LIN {X 0,Y 361.99,Z 158.394,A -85,B 0,C 180,E1 -12970.064,E2 -12970.064} C_VEL
LIN {X 0,Y 361.976,Z 158.397,A -85,B 0,C 180,E1 -12973.887,E2 -12973.887} C_VEL
LIN {X 0,Y 361.88,Z 158.406,A -85,B 0,C 180,E1 -12978.104,E2 -12978.104} C_VEL
LIN {X 0,Y 361.849,Z 158.413,A -85,B 0,C 180,E1 -12981.656,E2 -12981.656} C_VEL
LIN {X 0,Y 361.849,Z 158.412,A -85,B 0,C 180,E1 -12985.296,E2 -12985.296} C_VEL
LIN {X 0,Y 361.853,Z 158.41,A -85,B 0,C 180,E1 -12989.074,E2 -12989.074} C_VEL
LIN {X 0,Y 361.845,Z 158.411,A -85,B 0,C 180,E1 -12992.946,E2 -12992.946} C_VEL
LIN {X 0,Y 361.861,Z 158.409,A -85,B 0,C 180,E1 -12995.638,E2 -12995.638} C_VEL
LIN {X 0,Y 361.823,Z 158.416,A -85,B 0,C 180,E1 -12999.018,E2 -12999.018} C_VEL
LIN {X 0,Y 361.828,Z 158.414,A -85,B 0,C 180,E1 -13002.831,E2 -13002.831} C_VEL
LIN {X 0,Y 361.812,Z 158.413,A -85,B 0,C 180,E1 -13005.948,E2 -13005.948} C_VEL
LIN {X 0,Y 361.81,Z 158.416,A -85,B 0,C 180,E1 -13009.25,E2 -13009.25} C_VEL
LIN {X 0,Y 361.861,Z 158.412,A -85,B 0,C 180,E1 -13012.982,E2 -13012.982} C_VEL
LIN {X 0,Y 361.858,Z 158.412,A -85,B 0,C 180,E1 -13016.632,E2 -13016.632} C_VEL
LIN {X 0,Y 361.865,Z 158.409,A -85,B 0,C 180,E1 -13020.315,E2 -13020.315} C_VEL
LIN {X 0,Y 361.868,Z 158.547,A -85,B 0,C 180,E1 -13020.81,E2 -13020.81} C_VEL
LIN {X 0,Y 364.371,Z 170.848,A -85,B 0,C 180,E1 -13023.973,E2 -13023.973} C_VEL
LIN {X 0,Y 365.33,Z 177.294,A -85,B 0,C 180,E1 -13025.569,E2 -13025.569} C_VEL
LIN {X 0,Y 364.23,Z 189.968,A -85,B 0,C 180,E1 -13028.493,E2 -13028.493} C_VEL
LIN {X 0,Y 369.048,Z 223.646,A -85,B 0,C 180,E1 -13029.496,E2 -13029.496} C_VEL
LIN {X 0,Y 367.536,Z 298.731,A -85,B 0,C 180,E1 -13031.102,E2 -13031.102} C_VEL
LIN {X 0,Y 366.947,Z 312.235,A -85,B 0,C 180,E1 -13031.614,E2 -13031.614} C_VEL
LIN {X 0,Y 366.191,Z 324.024,A -85,B 0,C 180,E1 -13032.261,E2 -13032.261} C_VEL
LIN {X 0,Y 365.354,Z 335.279,A -85,B 0,C 180,E1 -13033.085,E2 -13033.085} C_VEL
LIN {X 0,Y 364.275,Z 346.955,A -85,B 0,C 180,E1 -13034.186,E2 -13034.186} C_VEL
LIN {X 0,Y 363.436,Z 357.505,A -85,B 0,C 180,E1 -13035.44,E2 -13035.44} C_VEL
LIN {X 0,Y 362.593,Z 366.984,A -85,B 0,C 180,E1 -13036.836,E2 -13036.836} C_VEL
LIN {X 0,Y 361.669,Z 376.126,A -85,B 0,C 180,E1 -13038.511,E2 -13038.511} C_VEL
LIN {X 0,Y 361.112,Z 383.491,A -85,B 0,C 180,E1 -13040.195,E2 -13040.195} C_VEL
LIN {X 0,Y 360.759,Z 388.451,A -85,B 0,C 180,E1 -13041.598,E2 -13041.598} C_VEL
LIN {X 0,Y 360.499,Z 393.254,A -85,B 0,C 180,E1 -13043.283,E2 -13043.283} C_VEL
LIN {X 0,Y 360.345,Z 396.905,A -85,B 0,C 180,E1 -13044.965,E2 -13044.965} C_VEL
LIN {X 0,Y 360.301,Z 399.51,A -85,B 0,C 180,E1 -13046.645,E2 -13046.645} C_VEL
LIN {X 0,Y 360.266,Z 400.723,A -85,B 0,C 180,E1 -13047.764,E2 -13047.764} C_VEL
LIN {X 0,Y 360.319,Z 401.482,A -85,B 0,C 180,E1 -13048.882,E2 -13048.882} C_VEL
LIN {X 0,Y 360.361,Z 401.829,A -85,B 0,C 180,E1 -13050,E2 -13050} C_VEL
LIN {X 0,Y 360.303,Z 401.777,A -85,B 0,C 180,E1 -13051.117,E2 -13051.117} C_VEL
LIN {X 0,Y 360.263,Z 401.326,A -85,B 0,C 180,E1 -13052.236,E2 -13052.236} C_VEL
LIN {X 0,Y 360.297,Z 400.429,A -85,B 0,C 180,E1 -13053.355,E2 -13053.355} C_VEL
LIN {X 0,Y 360.346,Z 399.119,A -85,B 0,C 180,E1 -13054.474,E2 -13054.474} C_VEL
LIN {X 0,Y 360.379,Z 396.74,A -85,B 0,C 180,E1 -13055.961,E2 -13055.961} C_VEL
LIN {X 0,Y 360.69,Z 392.557,A -85,B 0,C 180,E1 -13057.839,E2 -13057.839} C_VEL
LIN {X 0,Y 361.118,Z 387.637,A -85,B 0,C 180,E1 -13059.522,E2 -13059.522} C_VEL
LIN {X 0,Y 361.758,Z 381.447,A -85,B 0,C 180,E1 -13061.202,E2 -13061.202} C_VEL
LIN {X 0,Y 362.725,Z 373.766,A -85,B 0,C 180,E1 -13062.874,E2 -13062.874} C_VEL
LIN {X 0,Y 363.683,Z 365.931,A -85,B 0,C 180,E1 -13064.263,E2 -13064.263} C_VEL
LIN {X 0,Y 364.646,Z 356.392,A -85,B 0,C 180,E1 -13065.654,E2 -13065.654} C_VEL
LIN {X 0,Y 365.843,Z 345.844,A -85,B 0,C 180,E1 -13066.891,E2 -13066.891} C_VEL
LIN {X 0,Y 367.109,Z 334.15,A -85,B 0,C 180,E1 -13067.98,E2 -13067.98} C_VEL
LIN {X 0,Y 368.232,Z 321.75,A -85,B 0,C 180,E1 -13068.86,E2 -13068.86} C_VEL
LIN {X 0,Y 369.141,Z 308.873,A -85,B 0,C 180,E1 -13069.534,E2 -13069.534} C_VEL
LIN {X 0,Y 369.816,Z 296.528,A -85,B 0,C 180,E1 -13069.967,E2 -13069.967} C_VEL
LIN {X 0,Y 371.47,Z 222.319,A -85,B 0,C 180,E1 -13071.596,E2 -13071.596} C_VEL
LIN {X 0,Y 368.034,Z 201.179,A -85,B 0,C 180,E1 -13072.355,E2 -13072.355} C_VEL
LIN {X 0,Y 365.368,Z 188.435,A -85,B 0,C 180,E1 -13072.904,E2 -13072.904} C_VEL
LIN {X 0,Y 366.207,Z 179.523,A -85,B 0,C 180,E1 -13074.974,E2 -13074.974} C_VEL
LIN {X 0,Y 364.952,Z 172.094,A -85,B 0,C 180,E1 -13076.897,E2 -13076.897} C_VEL
LIN {X 0,Y 362.672,Z 161.769,A -85,B 0,C 180,E1 -13079.712,E2 -13079.712} C_VEL
LIN {X 0,Y 361.872,Z 158.417,A -85,B 0,C 180,E1 -13080.707,E2 -13080.707} C_VEL
LIN {X 0,Y 361.849,Z 158.412,A -85,B 0,C 180,E1 -13084.28,E2 -13084.28} C_VEL
LIN {X 0,Y 361.855,Z 158.414,A -85,B 0,C 180,E1 -13087.22,E2 -13087.22} C_VEL
LIN {X 0,Y 361.808,Z 158.419,A -85,B 0,C 180,E1 -13090.75,E2 -13090.75} C_VEL
LIN {X 0,Y 361.809,Z 158.42,A -85,B 0,C 180,E1 -13094.369,E2 -13094.369} C_VEL
LIN {X 0,Y 361.819,Z 158.411,A -85,B 0,C 180,E1 -13097.57,E2 -13097.57} C_VEL
LIN {X 0,Y 361.838,Z 158.412,A -85,B 0,C 180,E1 -13101.571,E2 -13101.571} C_VEL
LIN {X 0,Y 361.866,Z 158.409,A -85,B 0,C 180,E1 -13104.656,E2 -13104.656} C_VEL
LIN {X 0,Y 361.833,Z 158.413,A -85,B 0,C 180,E1 -13108.37,E2 -13108.37} C_VEL
LIN {X 0,Y 361.845,Z 158.41,A -85,B 0,C 180,E1 -13110.95,E2 -13110.95} C_VEL
LIN {X 0,Y 361.855,Z 158.409,A -85,B 0,C 180,E1 -13114.704,E2 -13114.704} C_VEL
LIN {X 0,Y 361.847,Z 158.408,A -85,B 0,C 180,E1 -13118.344,E2 -13118.344} C_VEL
LIN {X 0,Y 361.89,Z 158.402,A -85,B 0,C 180,E1 -13122.097,E2 -13122.097} C_VEL
LIN {X 0,Y 361.974,Z 158.395,A -85,B 0,C 180,E1 -13126.113,E2 -13126.113} C_VEL
LIN {X 0,Y 361.988,Z 158.395,A -85,B 0,C 180,E1 -13129.936,E2 -13129.936} C_VEL
LIN {X 0,Y 362.111,Z 158.378,A -85,B 0,C 180,E1 -13133.312,E2 -13133.312} C_VEL
LIN {X 0,Y 362.256,Z 158.359,A -85,B 0,C 180,E1 -13137.776,E2 -13137.776} C_VEL
LIN {X 0,Y 362.166,Z 158.367,A -85,B 0,C 180,E1 -13141.111,E2 -13141.111} C_VEL
LIN {X 0,Y 362.256,Z 158.362,A -85,B 0,C 180,E1 -13142.223,E2 -13142.223} C_VEL
LIN {X 0,Y 362.111,Z 158.379,A -85,B 0,C 180,E1 -13146.687,E2 -13146.687} C_VEL
LIN {X 0,Y 361.987,Z 158.399,A -85,B 0,C 180,E1 -13150.063,E2 -13150.063} C_VEL
LIN {X 0,Y 361.972,Z 158.404,A -85,B 0,C 180,E1 -13153.886,E2 -13153.886} C_VEL
LIN {X 0,Y 361.928,Z 158.506,A -85,B 0,C 180,E1 -13157.348,E2 -13157.348} C_VEL
LIN {X 0,Y 364.483,Z 169.841,A -85,B 0,C 180,E1 -13160.603,E2 -13160.603} C_VEL
LIN {X 0,Y 364.864,Z 171.752,A -85,B 0,C 180,E1 -13161.134,E2 -13161.134} C_VEL
LIN {X 0,Y 368.482,Z 181.215,A -85,B 0,C 180,E1 -13161.661,E2 -13161.661} C_VEL
LIN {X 0,Y 372.141,Z 198.437,A -85,B 0,C 180,E1 -13162.349,E2 -13162.349} C_VEL
LIN {X 0,Y 370.023,Z 279.828,A -85,B 0,C 180,E1 -13164.135,E2 -13164.135} C_VEL
LIN {X 0,Y 369.348,Z 293.268,A -85,B 0,C 180,E1 -13164.651,E2 -13164.651} C_VEL
LIN {X 0,Y 368.609,Z 305.305,A -85,B 0,C 180,E1 -13165.327,E2 -13165.327} C_VEL
LIN {X 0,Y 367.629,Z 317.028,A -85,B 0,C 180,E1 -13166.207,E2 -13166.207} C_VEL
LIN {X 0,Y 366.407,Z 329.368,A -85,B 0,C 180,E1 -13167.409,E2 -13167.409} C_VEL
LIN {X 0,Y 365.378,Z 338.355,A -85,B 0,C 180,E1 -13168.501,E2 -13168.501} C_VEL
LIN {X 0,Y 364.251,Z 347.761,A -85,B 0,C 180,E1 -13169.901,E2 -13169.901} C_VEL
LIN {X 0,Y 363.096,Z 356.944,A -85,B 0,C 180,E1 -13171.61,E2 -13171.61} C_VEL
LIN {X 0,Y 362.288,Z 363.667,A -85,B 0,C 180,E1 -13173.166,E2 -13173.166} C_VEL
LIN {X 0,Y 361.625,Z 369.267,A -85,B 0,C 180,E1 -13174.77,E2 -13174.77} C_VEL
LIN {X 0,Y 361.125,Z 373.689,A -85,B 0,C 180,E1 -13176.363,E2 -13176.363} C_VEL
LIN {X 0,Y 360.619,Z 378.205,A -85,B 0,C 180,E1 -13178.582,E2 -13178.582} C_VEL
LIN {X 0,Y 360.314,Z 380.682,A -85,B 0,C 180,E1 -13180.475,E2 -13180.475} C_VEL
LIN {X 0,Y 360.144,Z 381.878,A -85,B 0,C 180,E1 -13182.138,E2 -13182.138} C_VEL
LIN {X 0,Y 360.085,Z 382.184,A -85,B 0,C 180,E1 -13183.769,E2 -13183.769} C_VEL
LIN {X 0,Y 360.121,Z 381.648,A -85,B 0,C 180,E1 -13185.368,E2 -13185.368} C_VEL
LIN {X 0,Y 360.235,Z 380.281,A -85,B 0,C 180,E1 -13186.936,E2 -13186.936} C_VEL
LIN {X 0,Y 360.343,Z 378.163,A -85,B 0,C 180,E1 -13188.462,E2 -13188.462} C_VEL
LIN {X 0,Y 360.592,Z 375.269,A -85,B 0,C 180,E1 -13189.972,E2 -13189.972} C_VEL
LIN {X 0,Y 360.967,Z 370.522,A -85,B 0,C 180,E1 -13191.819,E2 -13191.819} C_VEL
LIN {X 0,Y 361.507,Z 364.434,A -85,B 0,C 180,E1 -13193.635,E2 -13193.635} C_VEL
LIN {X 0,Y 362.075,Z 357.751,A -85,B 0,C 180,E1 -13195.221,E2 -13195.221} C_VEL
LIN {X 0,Y 362.882,Z 349.41,A -85,B 0,C 180,E1 -13196.813,E2 -13196.813} C_VEL
LIN {X 0,Y 363.728,Z 340.279,A -85,B 0,C 180,E1 -13198.23,E2 -13198.23} C_VEL
LIN {X 0,Y 364.703,Z 329.228,A -85,B 0,C 180,E1 -13199.613,E2 -13199.613} C_VEL
LIN {X 0,Y 365.524,Z 318.906,A -85,B 0,C 180,E1 -13200.641,E2 -13200.641} C_VEL
LIN {X 0,Y 366.325,Z 307.35,A -85,B 0,C 180,E1 -13201.553,E2 -13201.553} C_VEL
LIN {X 0,Y 367.059,Z 294.631,A -85,B 0,C 180,E1 -13202.312,E2 -13202.312} C_VEL
LIN {X 0,Y 367.556,Z 281.435,A -85,B 0,C 180,E1 -13202.852,E2 -13202.852} C_VEL
LIN {X 0,Y 368.043,Z 261.332,A -85,B 0,C 180,E1 -13203.324,E2 -13203.324} C_VEL
LIN {X 0,Y 369.26,Z 196.419,A -85,B 0,C 180,E1 -13204.695,E2 -13204.695} C_VEL
LIN {X 0,Y 364.638,Z 172.365,A -85,B 0,C 180,E1 -13205.477,E2 -13205.477} C_VEL
LIN {X 0,Y 364.263,Z 170.887,A -85,B 0,C 180,E1 -13205.569,E2 -13205.569} C_VEL
LIN {X 0,Y 361.88,Z 158.41,A -85,B 0,C 180,E1 -13209.027,E2 -13209.027} C_VEL
LIN {X 0,Y 361.885,Z 158.405,A -85,B 0,C 180,E1 -13213.064,E2 -13213.064} C_VEL
LIN {X 0,Y 361.995,Z 158.395,A -85,B 0,C 180,E1 -13216.528,E2 -13216.528} C_VEL
LIN {X 0,Y 361.991,Z 158.393,A -85,B 0,C 180,E1 -13219.937,E2 -13219.937} C_VEL
LIN {X 0,Y 362.118,Z 158.375,A -85,B 0,C 180,E1 -13223.313,E2 -13223.313} C_VEL
LIN {X 0,Y 362.26,Z 158.359,A -85,B 0,C 180,E1 -13227.777,E2 -13227.777} C_VEL
LIN {X 0,Y 362.17,Z 158.368,A -85,B 0,C 180,E1 -13231.112,E2 -13231.112} C_VEL
LIN {X 0,Y 362.254,Z 158.362,A -85,B 0,C 180,E1 -13232.224,E2 -13232.224} C_VEL
LIN {X 0,Y 362.115,Z 158.375,A -85,B 0,C 180,E1 -13236.687,E2 -13236.687} C_VEL
LIN {X 0,Y 361.991,Z 158.395,A -85,B 0,C 180,E1 -13240.063,E2 -13240.063} C_VEL
LIN {X 0,Y 361.957,Z 158.395,A -85,B 0,C 180,E1 -13240.68,E2 -13240.68} C_VEL
LIN {X 0,Y 361.281,Z 158.483,A -85,B 0,C 180,E1 -13241.61,E2 -13241.61} C_VEL
LIN {X 0,Y 358.414,Z 158.837,A -85,B 0,C 180,E1 -13243.121,E2 -13243.121} C_VEL
LIN {X 0,Y 355.982,Z 159.14,A -85,B 0,C 180,E1 -13244.344,E2 -13244.344} C_VEL
LIN {X 0,Y 354.928,Z 159.272,A -85,B 0,C 180,E1 -13245.29,E2 -13245.29} C_VEL
LIN {X 0,Y 354.836,Z 159.281,A -85,B 0,C 180,E1 -13245.611,E2 -13245.611} C_VEL
LIN {X 0,Y 354.821,Z 159.284,A -85,B 0,C 180,E1 -13248.476,E2 -13248.476} C_VEL
LIN {X 0,Y 354.802,Z 159.287,A -85,B 0,C 180,E1 -13252.108,E2 -13252.108} C_VEL
LIN {X 0,Y 354.791,Z 159.29,A -85,B 0,C 180,E1 -13255.836,E2 -13255.836} C_VEL
LIN {X 0,Y 354.789,Z 159.291,A -85,B 0,C 180,E1 -13259.684,E2 -13259.684} C_VEL
LIN {X 0,Y 354.782,Z 159.288,A -85,B 0,C 180,E1 -13262.334,E2 -13262.334} C_VEL
LIN {X 0,Y 354.817,Z 159.286,A -85,B 0,C 180,E1 -13265.699,E2 -13265.699} C_VEL
LIN {X 0,Y 354.764,Z 159.295,A -85,B 0,C 180,E1 -13269.412,E2 -13269.412} C_VEL
LIN {X 0,Y 354.776,Z 159.293,A -85,B 0,C 180,E1 -13272.866,E2 -13272.866} C_VEL
LIN {X 0,Y 354.757,Z 159.291,A -85,B 0,C 180,E1 -13276.103,E2 -13276.103} C_VEL
LIN {X 0,Y 354.759,Z 159.295,A -85,B 0,C 180,E1 -13279.176,E2 -13279.176} C_VEL
LIN {X 0,Y 354.793,Z 159.289,A -85,B 0,C 180,E1 -13282.405,E2 -13282.405} C_VEL
LIN {X 0,Y 354.803,Z 159.291,A -85,B 0,C 180,E1 -13284.94,E2 -13284.94} C_VEL
LIN {X 0,Y 354.788,Z 159.29,A -85,B 0,C 180,E1 -13288.406,E2 -13288.406} C_VEL
LIN {X 0,Y 354.791,Z 159.287,A -85,B 0,C 180,E1 -13291.614,E2 -13291.614} C_VEL
LIN {X 0,Y 354.799,Z 159.287,A -85,B 0,C 180,E1 -13295.42,E2 -13295.42} C_VEL
LIN {X 0,Y 354.815,Z 159.285,A -85,B 0,C 180,E1 -13299.113,E2 -13299.113} C_VEL
LIN {X 0,Y 354.846,Z 159.284,A -85,B 0,C 180,E1 -13302.718,E2 -13302.718} C_VEL
LIN {X 0,Y 354.934,Z 159.274,A -85,B 0,C 180,E1 -13306.255,E2 -13306.255} C_VEL
LIN {X 0,Y 354.945,Z 159.269,A -85,B 0,C 180,E1 -13309.735,E2 -13309.735} C_VEL
LIN {X 0,Y 355.079,Z 159.251,A -85,B 0,C 180,E1 -13313.18,E2 -13313.18} C_VEL
LIN {X 0,Y 355.214,Z 159.237,A -85,B 0,C 180,E1 -13317.733,E2 -13317.733} C_VEL
LIN {X 0,Y 355.139,Z 159.244,A -85,B 0,C 180,E1 -13321.134,E2 -13321.134} C_VEL
LIN {X 0,Y 355.214,Z 159.238,A -85,B 0,C 180,E1 -13322.268,E2 -13322.268} C_VEL
LIN {X 0,Y 355.08,Z 159.251,A -85,B 0,C 180,E1 -13326.821,E2 -13326.821} C_VEL
LIN {X 0,Y 354.947,Z 159.27,A -85,B 0,C 180,E1 -13330.265,E2 -13330.265} C_VEL
LIN {X 0,Y 354.919,Z 159.275,A -85,B 0,C 180,E1 -13334.006,E2 -13334.006} C_VEL
LIN {X 0,Y 354.838,Z 159.284,A -85,B 0,C 180,E1 -13338.068,E2 -13338.068} C_VEL
LIN {X 0,Y 354.802,Z 159.287,A -85,B 0,C 180,E1 -13342.109,E2 -13342.109} C_VEL
LIN {X 0,Y 354.792,Z 159.29,A -85,B 0,C 180,E1 -13345.836,E2 -13345.836} C_VEL
LIN {X 0,Y 354.791,Z 159.291,A -85,B 0,C 180,E1 -13349.685,E2 -13349.685} C_VEL
LIN {X 0,Y 354.784,Z 159.288,A -85,B 0,C 180,E1 -13352.334,E2 -13352.334} C_VEL
LIN {X 0,Y 354.816,Z 159.286,A -85,B 0,C 180,E1 -13355.699,E2 -13355.699} C_VEL
LIN {X 0,Y 354.767,Z 159.294,A -85,B 0,C 180,E1 -13359.413,E2 -13359.413} C_VEL
LIN {X 0,Y 354.78,Z 159.292,A -85,B 0,C 180,E1 -13362.866,E2 -13362.866} C_VEL
LIN {X 0,Y 354.761,Z 159.291,A -85,B 0,C 180,E1 -13366.103,E2 -13366.103} C_VEL
LIN {X 0,Y 354.763,Z 159.295,A -85,B 0,C 180,E1 -13369.176,E2 -13369.176} C_VEL
LIN {X 0,Y 354.798,Z 159.288,A -85,B 0,C 180,E1 -13372.405,E2 -13372.405} C_VEL
LIN {X 0,Y 354.808,Z 159.29,A -85,B 0,C 180,E1 -13374.941,E2 -13374.941} C_VEL
LIN {X 0,Y 354.777,Z 159.292,A -85,B 0,C 180,E1 -13378.41,E2 -13378.41} C_VEL
LIN {X 0,Y 354.843,Z 159.471,A -85,B 0,C 180,E1 -13380.537,E2 -13380.537} C_VEL
LIN {X 0,Y 357.324,Z 171.644,A -85,B 0,C 180,E1 -13383.734,E2 -13383.734} C_VEL
LIN {X 0,Y 358.37,Z 178.159,A -85,B 0,C 180,E1 -13385.382,E2 -13385.382} C_VEL
LIN {X 0,Y 357.308,Z 189.781,A -85,B 0,C 180,E1 -13388.119,E2 -13388.119} C_VEL
LIN {X 0,Y 362.287,Z 224.115,A -85,B 0,C 180,E1 -13389.17,E2 -13389.17} C_VEL
LIN {X 0,Y 360.705,Z 298.839,A -85,B 0,C 180,E1 -13390.805,E2 -13390.805} C_VEL
LIN {X 0,Y 360.103,Z 312.238,A -85,B 0,C 180,E1 -13391.325,E2 -13391.325} C_VEL
LIN {X 0,Y 359.22,Z 325.018,A -85,B 0,C 180,E1 -13392.053,E2 -13392.053} C_VEL
LIN {X 0,Y 358.219,Z 337.567,A -85,B 0,C 180,E1 -13393.032,E2 -13393.032} C_VEL
LIN {X 0,Y 357.18,Z 348.783,A -85,B 0,C 180,E1 -13394.155,E2 -13394.155} C_VEL
LIN {X 0,Y 356.337,Z 358.927,A -85,B 0,C 180,E1 -13395.436,E2 -13395.436} C_VEL
LIN {X 0,Y 355.495,Z 368.09,A -85,B 0,C 180,E1 -13396.859,E2 -13396.859} C_VEL
LIN {X 0,Y 354.53,Z 377.017,A -85,B 0,C 180,E1 -13398.566,E2 -13398.566} C_VEL
LIN {X 0,Y 353.987,Z 384.141,A -85,B 0,C 180,E1 -13400.284,E2 -13400.284} C_VEL
LIN {X 0,Y 353.577,Z 389.819,A -85,B 0,C 180,E1 -13402.002,E2 -13402.002} C_VEL
LIN {X 0,Y 353.318,Z 394.95,A -85,B 0,C 180,E1 -13404.031,E2 -13404.031} C_VEL
LIN {X 0,Y 353.276,Z 397.597,A -85,B 0,C 180,E1 -13405.436,E2 -13405.436} C_VEL
LIN {X 0,Y 353.223,Z 399.243,A -85,B 0,C 180,E1 -13406.578,E2 -13406.578} C_VEL
LIN {X 0,Y 353.175,Z 400.475,A -85,B 0,C 180,E1 -13407.719,E2 -13407.719} C_VEL
LIN {X 0,Y 353.219,Z 401.263,A -85,B 0,C 180,E1 -13408.86,E2 -13408.86} C_VEL
LIN {X 0,Y 353.263,Z 401.625,A -85,B 0,C 180,E1 -13410,E2 -13410} C_VEL
LIN {X 0,Y 353.203,Z 401.586,A -85,B 0,C 180,E1 -13411.14,E2 -13411.14} C_VEL
LIN {X 0,Y 353.171,Z 401.154,A -85,B 0,C 180,E1 -13412.281,E2 -13412.281} C_VEL
LIN {X 0,Y 353.218,Z 400.284,A -85,B 0,C 180,E1 -13413.422,E2 -13413.422} C_VEL
LIN {X 0,Y 353.26,Z 398.991,A -85,B 0,C 180,E1 -13414.564,E2 -13414.564} C_VEL
LIN {X 0,Y 353.277,Z 396.97,A -85,B 0,C 180,E1 -13415.904,E2 -13415.904} C_VEL
LIN {X 0,Y 353.63,Z 392.507,A -85,B 0,C 180,E1 -13417.996,E2 -13417.996} C_VEL
LIN {X 0,Y 354.079,Z 387.624,A -85,B 0,C 180,E1 -13419.713,E2 -13419.713} C_VEL
LIN {X 0,Y 354.761,Z 381.471,A -85,B 0,C 180,E1 -13421.426,E2 -13421.426} C_VEL
LIN {X 0,Y 355.795,Z 373.833,A -85,B 0,C 180,E1 -13423.129,E2 -13423.129} C_VEL
LIN {X 0,Y 356.788,Z 366.054,A -85,B 0,C 180,E1 -13424.545,E2 -13424.545} C_VEL
LIN {X 0,Y 357.807,Z 356.601,A -85,B 0,C 180,E1 -13425.961,E2 -13425.961} C_VEL
LIN {X 0,Y 359.061,Z 346.145,A -85,B 0,C 180,E1 -13427.22,E2 -13427.22} C_VEL
LIN {X 0,Y 360.389,Z 334.612,A -85,B 0,C 180,E1 -13428.328,E2 -13428.328} C_VEL
LIN {X 0,Y 361.545,Z 322.521,A -85,B 0,C 180,E1 -13429.222,E2 -13429.222} C_VEL
LIN {X 0,Y 362.568,Z 309.287,A -85,B 0,C 180,E1 -13429.94,E2 -13429.94} C_VEL
LIN {X 0,Y 363.309,Z 296.322,A -85,B 0,C 180,E1 -13430.411,E2 -13430.411} C_VEL
LIN {X 0,Y 365.049,Z 223.186,A -85,B 0,C 180,E1 -13432.049,E2 -13432.049} C_VEL
LIN {X 0,Y 361.717,Z 202.801,A -85,B 0,C 180,E1 -13432.805,E2 -13432.805} C_VEL
LIN {X 0,Y 358.674,Z 188.33,A -85,B 0,C 180,E1 -13433.423,E2 -13433.423} C_VEL
LIN {X 0,Y 359.378,Z 180.984,A -85,B 0,C 180,E1 -13435.172,E2 -13435.172} C_VEL
LIN {X 0,Y 357.929,Z 172.952,A -85,B 0,C 180,E1 -13437.306,E2 -13437.306} C_VEL
LIN {X 0,Y 355.615,Z 162.455,A -85,B 0,C 180,E1 -13440.261,E2 -13440.261} C_VEL
LIN {X 0,Y 354.789,Z 159.299,A -85,B 0,C 180,E1 -13441.216,E2 -13441.216} C_VEL
LIN {X 0,Y 354.807,Z 159.29,A -85,B 0,C 180,E1 -13445.059,E2 -13445.059} C_VEL
LIN {X 0,Y 354.791,Z 159.293,A -85,B 0,C 180,E1 -13447.884,E2 -13447.884} C_VEL
LIN {X 0,Y 354.765,Z 159.299,A -85,B 0,C 180,E1 -13451.167,E2 -13451.167} C_VEL
LIN {X 0,Y 354.755,Z 159.298,A -85,B 0,C 180,E1 -13454.504,E2 -13454.504} C_VEL
LIN {X 0,Y 354.778,Z 159.288,A -85,B 0,C 180,E1 -13457.66,E2 -13457.66} C_VEL
LIN {X 0,Y 354.782,Z 159.288,A -85,B 0,C 180,E1 -13460.661,E2 -13460.661} C_VEL
LIN {X 0,Y 354.814,Z 159.284,A -85,B 0,C 180,E1 -13464.301,E2 -13464.301} C_VEL
LIN {X 0,Y 354.782,Z 159.288,A -85,B 0,C 180,E1 -13467.666,E2 -13467.666} C_VEL
LIN {X 0,Y 354.784,Z 159.289,A -85,B 0,C 180,E1 -13471.613,E2 -13471.613} C_VEL
LIN {X 0,Y 354.799,Z 159.289,A -85,B 0,C 180,E1 -13475.419,E2 -13475.419} C_VEL
LIN {X 0,Y 354.813,Z 159.287,A -85,B 0,C 180,E1 -13479.112,E2 -13479.112} C_VEL
LIN {X 0,Y 354.833,Z 159.286,A -85,B 0,C 180,E1 -13482.716,E2 -13482.716} C_VEL
LIN {X 0,Y 354.933,Z 159.273,A -85,B 0,C 180,E1 -13486.254,E2 -13486.254} C_VEL
LIN {X 0,Y 354.944,Z 159.27,A -85,B 0,C 180,E1 -13489.734,E2 -13489.734} C_VEL
LIN {X 0,Y 355.078,Z 159.254,A -85,B 0,C 180,E1 -13493.179,E2 -13493.179} C_VEL
LIN {X 0,Y 355.218,Z 159.236,A -85,B 0,C 180,E1 -13497.732,E2 -13497.732} C_VEL
LIN {X 0,Y 355.137,Z 159.243,A -85,B 0,C 180,E1 -13501.133,E2 -13501.133} C_VEL
LIN {X 0,Y 355.218,Z 159.239,A -85,B 0,C 180,E1 -13502.267,E2 -13502.267} C_VEL
LIN {X 0,Y 355.077,Z 159.255,A -85,B 0,C 180,E1 -13506.82,E2 -13506.82} C_VEL
LIN {X 0,Y 354.944,Z 159.278,A -85,B 0,C 180,E1 -13510.265,E2 -13510.265} C_VEL
LIN {X 0,Y 354.916,Z 159.283,A -85,B 0,C 180,E1 -13514.005,E2 -13514.005} C_VEL
LIN {X 0,Y 354.879,Z 159.436,A -85,B 0,C 180,E1 -13516.835,E2 -13516.835} C_VEL
LIN {X 0,Y 357.426,Z 170.546,A -85,B 0,C 180,E1 -13520.126,E2 -13520.126} C_VEL
LIN {X 0,Y 357.766,Z 172.076,A -85,B 0,C 180,E1 -13520.556,E2 -13520.556} C_VEL
LIN {X 0,Y 362.311,Z 183.376,A -85,B 0,C 180,E1 -13521.223,E2 -13521.223} C_VEL
LIN {X 0,Y 365.726,Z 199.169,A -85,B 0,C 180,E1 -13521.882,E2 -13521.882} C_VEL
LIN {X 0,Y 363.518,Z 280.444,A -85,B 0,C 180,E1 -13523.707,E2 -13523.707} C_VEL
LIN {X 0,Y 362.819,Z 293.51,A -85,B 0,C 180,E1 -13524.22,E2 -13524.22} C_VEL
LIN {X 0,Y 362.008,Z 306.066,A -85,B 0,C 180,E1 -13524.945,E2 -13524.945} C_VEL
LIN {X 0,Y 361.032,Z 317.023,A -85,B 0,C 180,E1 -13525.785,E2 -13525.785} C_VEL
LIN {X 0,Y 359.944,Z 327.832,A -85,B 0,C 180,E1 -13526.841,E2 -13526.841} C_VEL
LIN {X 0,Y 358.626,Z 338.491,A -85,B 0,C 180,E1 -13528.134,E2 -13528.134} C_VEL
LIN {X 0,Y 357.574,Z 347.133,A -85,B 0,C 180,E1 -13529.43,E2 -13529.43} C_VEL
LIN {X 0,Y 356.383,Z 356.109,A -85,B 0,C 180,E1 -13531.091,E2 -13531.091} C_VEL
LIN {X 0,Y 355.328,Z 364.097,A -85,B 0,C 180,E1 -13532.95,E2 -13532.95} C_VEL
LIN {X 0,Y 354.57,Z 370.126,A -85,B 0,C 180,E1 -13534.739,E2 -13534.739} C_VEL
LIN {X 0,Y 353.995,Z 374.842,A -85,B 0,C 180,E1 -13536.555,E2 -13536.555} C_VEL
LIN {X 0,Y 353.633,Z 377.793,A -85,B 0,C 180,E1 -13538.03,E2 -13538.03} C_VEL
LIN {X 0,Y 353.343,Z 379.99,A -85,B 0,C 180,E1 -13539.529,E2 -13539.529} C_VEL
LIN {X 0,Y 353.145,Z 381.497,A -85,B 0,C 180,E1 -13541.051,E2 -13541.051} C_VEL
LIN {X 0,Y 353.011,Z 382.298,A -85,B 0,C 180,E1 -13542.601,E2 -13542.601} C_VEL
LIN {X 0,Y 352.991,Z 382.298,A -85,B 0,C 180,E1 -13544.214,E2 -13544.214} C_VEL
LIN {X 0,Y 353.051,Z 381.485,A -85,B 0,C 180,E1 -13545.836,E2 -13545.836} C_VEL
LIN {X 0,Y 353.176,Z 379.896,A -85,B 0,C 180,E1 -13547.424,E2 -13547.424} C_VEL
LIN {X 0,Y 353.334,Z 377.33,A -85,B 0,C 180,E1 -13549.098,E2 -13549.098} C_VEL
LIN {X 0,Y 353.67,Z 373.695,A -85,B 0,C 180,E1 -13550.804,E2 -13550.804} C_VEL
LIN {X 0,Y 354.076,Z 368.782,A -85,B 0,C 180,E1 -13552.556,E2 -13552.556} C_VEL
LIN {X 0,Y 354.6,Z 362.363,A -85,B 0,C 180,E1 -13554.35,E2 -13554.35} C_VEL
LIN {X 0,Y 355.403,Z 354.222,A -85,B 0,C 180,E1 -13556.153,E2 -13556.153} C_VEL
LIN {X 0,Y 356.388,Z 344.609,A -85,B 0,C 180,E1 -13557.83,E2 -13557.83} C_VEL
LIN {X 0,Y 357.322,Z 334.559,A -85,B 0,C 180,E1 -13559.245,E2 -13559.245} C_VEL
LIN {X 0,Y 358.289,Z 323.39,A -85,B 0,C 180,E1 -13560.494,E2 -13560.494} C_VEL
LIN {X 0,Y 359.139,Z 312.278,A -85,B 0,C 180,E1 -13561.48,E2 -13561.48} C_VEL
LIN {X 0,Y 359.973,Z 300.386,A -85,B 0,C 180,E1 -13562.296,E2 -13562.296} C_VEL
LIN {X 0,Y 360.548,Z 287.626,A -85,B 0,C 180,E1 -13562.934,E2 -13562.934} C_VEL
LIN {X 0,Y 361.007,Z 274.257,A -85,B 0,C 180,E1 -13563.362,E2 -13563.362} C_VEL
LIN {X 0,Y 362.523,Z 197.44,A -85,B 0,C 180,E1 -13565.019,E2 -13565.019} C_VEL
LIN {X 0,Y 358.133,Z 174.479,A -85,B 0,C 180,E1 -13565.779,E2 -13565.779} C_VEL
LIN {X 0,Y 357.111,Z 171.135,A -85,B 0,C 180,E1 -13565.937,E2 -13565.937} C_VEL
LIN {X 0,Y 354.827,Z 159.287,A -85,B 0,C 180,E1 -13569.303,E2 -13569.303} C_VEL
LIN {X 0,Y 354.847,Z 159.284,A -85,B 0,C 180,E1 -13572.718,E2 -13572.718} C_VEL
LIN {X 0,Y 354.936,Z 159.274,A -85,B 0,C 180,E1 -13576.255,E2 -13576.255} C_VEL
LIN {X 0,Y 354.947,Z 159.269,A -85,B 0,C 180,E1 -13579.735,E2 -13579.735} C_VEL
LIN {X 0,Y 355.083,Z 159.251,A -85,B 0,C 180,E1 -13583.18,E2 -13583.18} C_VEL
LIN {X 0,Y 355.222,Z 159.236,A -85,B 0,C 180,E1 -13587.732,E2 -13587.732} C_VEL
LIN {X 0,Y 355.141,Z 159.244,A -85,B 0,C 180,E1 -13591.134,E2 -13591.134} C_VEL
LIN {X 0,Y 355.216,Z 159.238,A -85,B 0,C 180,E1 -13592.268,E2 -13592.268} C_VEL
LIN {X 0,Y 355.081,Z 159.251,A -85,B 0,C 180,E1 -13596.82,E2 -13596.82} C_VEL
LIN {X 0,Y 354.948,Z 159.27,A -85,B 0,C 180,E1 -13600.265,E2 -13600.265} C_VEL
LIN {X 0,Y 354.919,Z 159.275,A -85,B 0,C 180,E1 -13604.006,E2 -13604.006} C_VEL
LIN {X 0,Y 354.836,Z 159.281,A -85,B 0,C 180,E1 -13605.611,E2 -13605.611} C_VEL
LIN {X 0,Y 354.149,Z 159.369,A -85,B 0,C 180,E1 -13606.559,E2 -13606.559} C_VEL
LIN {X 0,Y 351.278,Z 159.728,A -85,B 0,C 180,E1 -13608.1,E2 -13608.1} C_VEL
LIN {X 0,Y 348.859,Z 160.029,A -85,B 0,C 180,E1 -13609.347,E2 -13609.347} C_VEL
LIN {X 0,Y 347.828,Z 160.156,A -85,B 0,C 180,E1 -13610.312,E2 -13610.312} C_VEL
LIN {X 0,Y 347.748,Z 160.165,A -85,B 0,C 180,E1 -13610.639,E2 -13610.639} C_VEL
LIN {X 0,Y 347.765,Z 160.162,A -85,B 0,C 180,E1 -13614.578,E2 -13614.578} C_VEL
LIN {X 0,Y 347.721,Z 160.172,A -85,B 0,C 180,E1 -13617.701,E2 -13617.701} C_VEL
LIN {X 0,Y 347.732,Z 160.167,A -85,B 0,C 180,E1 -13620.349,E2 -13620.349} C_VEL
LIN {X 0,Y 347.744,Z 160.166,A -85,B 0,C 180,E1 -13624.044,E2 -13624.044} C_VEL
LIN {X 0,Y 347.751,Z 160.17,A -85,B 0,C 180,E1 -13627.322,E2 -13627.322} C_VEL
LIN {X 0,Y 347.691,Z 160.172,A -85,B 0,C 180,E1 -13630.302,E2 -13630.302} C_VEL
LIN {X 0,Y 347.716,Z 160.172,A -85,B 0,C 180,E1 -13633.409,E2 -13633.409} C_VEL
LIN {X 0,Y 347.718,Z 160.171,A -85,B 0,C 180,E1 -13636.687,E2 -13636.687} C_VEL
LIN {X 0,Y 347.696,Z 160.171,A -85,B 0,C 180,E1 -13640.182,E2 -13640.182} C_VEL
LIN {X 0,Y 347.749,Z 160.168,A -85,B 0,C 180,E1 -13642.678,E2 -13642.678} C_VEL
LIN {X 0,Y 347.743,Z 160.165,A -85,B 0,C 180,E1 -13645.957,E2 -13645.957} C_VEL
LIN {X 0,Y 347.733,Z 160.167,A -85,B 0,C 180,E1 -13649.651,E2 -13649.651} C_VEL
LIN {X 0,Y 347.729,Z 160.167,A -85,B 0,C 180,E1 -13653.6,E2 -13653.6} C_VEL
LIN {X 0,Y 347.743,Z 160.167,A -85,B 0,C 180,E1 -13656.159,E2 -13656.159} C_VEL
LIN {X 0,Y 347.766,Z 160.163,A -85,B 0,C 180,E1 -13659.907,E2 -13659.907} C_VEL
LIN {X 0,Y 347.792,Z 160.159,A -85,B 0,C 180,E1 -13663.567,E2 -13663.567} C_VEL
LIN {X 0,Y 347.879,Z 160.149,A -85,B 0,C 180,E1 -13667.161,E2 -13667.161} C_VEL
LIN {X 0,Y 347.928,Z 160.144,A -85,B 0,C 180,E1 -13670.701,E2 -13670.701} C_VEL
LIN {X 0,Y 348.03,Z 160.136,A -85,B 0,C 180,E1 -13674.206,E2 -13674.206} C_VEL
LIN {X 0,Y 348.176,Z 160.113,A -85,B 0,C 180,E1 -13677.687,E2 -13677.687} C_VEL
LIN {X 0,Y 348.111,Z 160.12,A -85,B 0,C 180,E1 -13681.157,E2 -13681.157} C_VEL
LIN {X 0,Y 348.176,Z 160.114,A -85,B 0,C 180,E1 -13682.314,E2 -13682.314} C_VEL
LIN {X 0,Y 348.047,Z 160.127,A -85,B 0,C 180,E1 -13686.959,E2 -13686.959} C_VEL
LIN {X 0,Y 347.887,Z 160.148,A -85,B 0,C 180,E1 -13690.476,E2 -13690.476} C_VEL
LIN {X 0,Y 347.877,Z 160.151,A -85,B 0,C 180,E1 -13694.138,E2 -13694.138} C_VEL
LIN {X 0,Y 347.789,Z 160.161,A -85,B 0,C 180,E1 -13698.241,E2 -13698.241} C_VEL
LIN {X 0,Y 347.76,Z 160.169,A -85,B 0,C 180,E1 -13701.625,E2 -13701.625} C_VEL
LIN {X 0,Y 347.731,Z 160.169,A -85,B 0,C 180,E1 -13705.115,E2 -13705.115} C_VEL
LIN {X 0,Y 347.722,Z 160.171,A -85,B 0,C 180,E1 -13707.702,E2 -13707.702} C_VEL
LIN {X 0,Y 347.733,Z 160.166,A -85,B 0,C 180,E1 -13710.35,E2 -13710.35} C_VEL
LIN {X 0,Y 347.746,Z 160.165,A -85,B 0,C 180,E1 -13714.044,E2 -13714.044} C_VEL
LIN {X 0,Y 347.753,Z 160.169,A -85,B 0,C 180,E1 -13717.323,E2 -13717.323} C_VEL
LIN {X 0,Y 347.695,Z 160.171,A -85,B 0,C 180,E1 -13720.303,E2 -13720.303} C_VEL
LIN {X 0,Y 347.72,Z 160.171,A -85,B 0,C 180,E1 -13723.409,E2 -13723.409} C_VEL
LIN {X 0,Y 347.722,Z 160.171,A -85,B 0,C 180,E1 -13726.688,E2 -13726.688} C_VEL
LIN {X 0,Y 347.701,Z 160.171,A -85,B 0,C 180,E1 -13730.183,E2 -13730.183} C_VEL
LIN {X 0,Y 347.754,Z 160.168,A -85,B 0,C 180,E1 -13732.679,E2 -13732.679} C_VEL
LIN {X 0,Y 347.749,Z 160.165,A -85,B 0,C 180,E1 -13735.957,E2 -13735.957} C_VEL
LIN {X 0,Y 347.771,Z 160.164,A -85,B 0,C 180,E1 -13740.152,E2 -13740.152} C_VEL
LIN {X 0,Y 350.263,Z 172.424,A -85,B 0,C 180,E1 -13743.484,E2 -13743.484} C_VEL
LIN {X 0,Y 351.376,Z 178.898,A -85,B 0,C 180,E1 -13745.164,E2 -13745.164} C_VEL
LIN {X 0,Y 350.401,Z 189.619,A -85,B 0,C 180,E1 -13747.739,E2 -13747.739} C_VEL
LIN {X 0,Y 355.512,Z 224.551,A -85,B 0,C 180,E1 -13748.837,E2 -13748.837} C_VEL
LIN {X 0,Y 353.88,Z 298.633,A -85,B 0,C 180,E1 -13750.495,E2 -13750.495} C_VEL
LIN {X 0,Y 353.27,Z 312.027,A -85,B 0,C 180,E1 -13751.026,E2 -13751.026} C_VEL
LIN {X 0,Y 352.35,Z 324.808,A -85,B 0,C 180,E1 -13751.766,E2 -13751.766} C_VEL
LIN {X 0,Y 351.421,Z 336.572,A -85,B 0,C 180,E1 -13752.694,E2 -13752.694} C_VEL
LIN {X 0,Y 350.283,Z 347.95,A -85,B 0,C 180,E1 -13753.836,E2 -13753.836} C_VEL
LIN {X 0,Y 349.399,Z 358.241,A -85,B 0,C 180,E1 -13755.14,E2 -13755.14} C_VEL
LIN {X 0,Y 348.511,Z 367.491,A -85,B 0,C 180,E1 -13756.591,E2 -13756.591} C_VEL
LIN {X 0,Y 347.536,Z 376.492,A -85,B 0,C 180,E1 -13758.333,E2 -13758.333} C_VEL
LIN {X 0,Y 346.946,Z 383.706,A -85,B 0,C 180,E1 -13760.085,E2 -13760.085} C_VEL
LIN {X 0,Y 346.524,Z 389.435,A -85,B 0,C 180,E1 -13761.838,E2 -13761.838} C_VEL
LIN {X 0,Y 346.295,Z 393.927,A -85,B 0,C 180,E1 -13763.592,E2 -13763.592} C_VEL
LIN {X 0,Y 346.17,Z 397.299,A -85,B 0,C 180,E1 -13765.342,E2 -13765.342} C_VEL
LIN {X 0,Y 346.147,Z 398.965,A -85,B 0,C 180,E1 -13766.508,E2 -13766.508} C_VEL
LIN {X 0,Y 346.086,Z 400.215,A -85,B 0,C 180,E1 -13767.672,E2 -13767.672} C_VEL
LIN {X 0,Y 346.119,Z 401.038,A -85,B 0,C 180,E1 -13768.836,E2 -13768.836} C_VEL
LIN {X 0,Y 346.166,Z 401.418,A -85,B 0,C 180,E1 -13770,E2 -13770} C_VEL
LIN {X 0,Y 346.104,Z 401.398,A -85,B 0,C 180,E1 -13771.163,E2 -13771.163} C_VEL
LIN {X 0,Y 346.082,Z 400.983,A -85,B 0,C 180,E1 -13772.327,E2 -13772.327} C_VEL
LIN {X 0,Y 346.141,Z 400.148,A -85,B 0,C 180,E1 -13773.492,E2 -13773.492} C_VEL
LIN {X 0,Y 346.158,Z 398.872,A -85,B 0,C 180,E1 -13774.658,E2 -13774.658} C_VEL
LIN {X 0,Y 346.243,Z 396.181,A -85,B 0,C 180,E1 -13776.409,E2 -13776.409} C_VEL
LIN {X 0,Y 346.573,Z 392.458,A -85,B 0,C 180,E1 -13778.16,E2 -13778.16} C_VEL
LIN {X 0,Y 347.057,Z 387.61,A -85,B 0,C 180,E1 -13779.911,E2 -13779.911} C_VEL
LIN {X 0,Y 347.769,Z 381.495,A -85,B 0,C 180,E1 -13781.659,E2 -13781.659} C_VEL
LIN {X 0,Y 348.859,Z 373.91,A -85,B 0,C 180,E1 -13783.395,E2 -13783.395} C_VEL
LIN {X 0,Y 349.9,Z 366.207,A -85,B 0,C 180,E1 -13784.838,E2 -13784.838} C_VEL
LIN {X 0,Y 350.999,Z 356.892,A -85,B 0,C 180,E1 -13786.279,E2 -13786.279} C_VEL
LIN {X 0,Y 352.305,Z 346.558,A -85,B 0,C 180,E1 -13787.561,E2 -13787.561} C_VEL
LIN {X 0,Y 353.693,Z 335.157,A -85,B 0,C 180,E1 -13788.687,E2 -13788.687} C_VEL
LIN {X 0,Y 354.893,Z 323.363,A -85,B 0,C 180,E1 -13789.597,E2 -13789.597} C_VEL
LIN {X 0,Y 355.957,Z 310.495,A -85,B 0,C 180,E1 -13790.326,E2 -13790.326} C_VEL
LIN {X 0,Y 356.766,Z 297.187,A -85,B 0,C 180,E1 -13790.84,E2 -13790.84} C_VEL
LIN {X 0,Y 358.707,Z 224.635,A -85,B 0,C 180,E1 -13792.5,E2 -13792.5} C_VEL
LIN {X 0,Y 355.52,Z 204.632,A -85,B 0,C 180,E1 -13793.268,E2 -13793.268} C_VEL
LIN {X 0,Y 352.018,Z 188.033,A -85,B 0,C 180,E1 -13794.019,E2 -13794.019} C_VEL
LIN {X 0,Y 352.542,Z 182.448,A -85,B 0,C 180,E1 -13795.379,E2 -13795.379} C_VEL
LIN {X 0,Y 350.527,Z 171.725,A -85,B 0,C 180,E1 -13798.335,E2 -13798.335} C_VEL
LIN {X 0,Y 348.082,Z 161.578,A -85,B 0,C 180,E1 -13801.325,E2 -13801.325} C_VEL
LIN {X 0,Y 347.733,Z 160.176,A -85,B 0,C 180,E1 -13801.806,E2 -13801.806} C_VEL
LIN {X 0,Y 347.742,Z 160.17,A -85,B 0,C 180,E1 -13804.463,E2 -13804.463} C_VEL
LIN {X 0,Y 347.76,Z 160.169,A -85,B 0,C 180,E1 -13807.985,E2 -13807.985} C_VEL
LIN {X 0,Y 347.738,Z 160.173,A -85,B 0,C 180,E1 -13811.831,E2 -13811.831} C_VEL
LIN {X 0,Y 347.697,Z 160.174,A -85,B 0,C 180,E1 -13815.027,E2 -13815.027} C_VEL
LIN {X 0,Y 347.735,Z 160.168,A -85,B 0,C 180,E1 -13818.399,E2 -13818.399} C_VEL
LIN {X 0,Y 347.758,Z 160.166,A -85,B 0,C 180,E1 -13822.013,E2 -13822.013} C_VEL
LIN {X 0,Y 347.739,Z 160.167,A -85,B 0,C 180,E1 -13825.535,E2 -13825.535} C_VEL
LIN {X 0,Y 347.74,Z 160.168,A -85,B 0,C 180,E1 -13828.299,E2 -13828.299} C_VEL
LIN {X 0,Y 347.736,Z 160.167,A -85,B 0,C 180,E1 -13830.983,E2 -13830.983} C_VEL
LIN {X 0,Y 347.729,Z 160.161,A -85,B 0,C 180,E1 -13833.599,E2 -13833.599} C_VEL
LIN {X 0,Y 347.743,Z 160.169,A -85,B 0,C 180,E1 -13836.158,E2 -13836.158} C_VEL
LIN {X 0,Y 347.759,Z 160.167,A -85,B 0,C 180,E1 -13839.906,E2 -13839.906} C_VEL
LIN {X 0,Y 347.781,Z 160.163,A -85,B 0,C 180,E1 -13843.565,E2 -13843.565} C_VEL
LIN {X 0,Y 347.878,Z 160.15,A -85,B 0,C 180,E1 -13847.16,E2 -13847.16} C_VEL
LIN {X 0,Y 347.927,Z 160.144,A -85,B 0,C 180,E1 -13850.7,E2 -13850.7} C_VEL
LIN {X 0,Y 348.028,Z 160.13,A -85,B 0,C 180,E1 -13854.205,E2 -13854.205} C_VEL
LIN {X 0,Y 348.18,Z 160.112,A -85,B 0,C 180,E1 -13857.686,E2 -13857.686} C_VEL
LIN {X 0,Y 348.109,Z 160.119,A -85,B 0,C 180,E1 -13861.156,E2 -13861.156} C_VEL
LIN {X 0,Y 348.179,Z 160.115,A -85,B 0,C 180,E1 -13862.313,E2 -13862.313} C_VEL
LIN {X 0,Y 348.044,Z 160.132,A -85,B 0,C 180,E1 -13866.958,E2 -13866.958} C_VEL
LIN {X 0,Y 347.884,Z 160.157,A -85,B 0,C 180,E1 -13870.475,E2 -13870.475} C_VEL
LIN {X 0,Y 347.873,Z 160.16,A -85,B 0,C 180,E1 -13874.137,E2 -13874.137} C_VEL
LIN {X 0,Y 347.814,Z 160.326,A -85,B 0,C 180,E1 -13876.281,E2 -13876.281} C_VEL
LIN {X 0,Y 349.748,Z 168.328,A -85,B 0,C 180,E1 -13878.754,E2 -13878.754} C_VEL
LIN {X 0,Y 350.595,Z 172.258,A -85,B 0,C 180,E1 -13879.924,E2 -13879.924} C_VEL
LIN {X 0,Y 356.344,Z 186.112,A -85,B 0,C 180,E1 -13880.793,E2 -13880.793} C_VEL
LIN {X 0,Y 359.314,Z 200.12,A -85,B 0,C 180,E1 -13881.398,E2 -13881.398} C_VEL
LIN {X 0,Y 357.034,Z 280.433,A -85,B 0,C 180,E1 -13883.241,E2 -13883.241} C_VEL
LIN {X 0,Y 356.306,Z 293.766,A -85,B 0,C 180,E1 -13883.773,E2 -13883.773} C_VEL
LIN {X 0,Y 355.406,Z 306.843,A -85,B 0,C 180,E1 -13884.548,E2 -13884.548} C_VEL
LIN {X 0,Y 354.247,Z 319.087,A -85,B 0,C 180,E1 -13885.531,E2 -13885.531} C_VEL
LIN {X 0,Y 353.17,Z 329.113,A -85,B 0,C 180,E1 -13886.555,E2 -13886.555} C_VEL
LIN {X 0,Y 351.835,Z 339.253,A -85,B 0,C 180,E1 -13887.825,E2 -13887.825} C_VEL
LIN {X 0,Y 350.664,Z 348.332,A -85,B 0,C 180,E1 -13889.243,E2 -13889.243} C_VEL
LIN {X 0,Y 349.457,Z 356.775,A -85,B 0,C 180,E1 -13890.865,E2 -13890.865} C_VEL
LIN {X 0,Y 348.458,Z 363.826,A -85,B 0,C 180,E1 -13892.541,E2 -13892.541} C_VEL
LIN {X 0,Y 347.587,Z 370.306,A -85,B 0,C 180,E1 -13894.481,E2 -13894.481} C_VEL
LIN {X 0,Y 346.861,Z 375.824,A -85,B 0,C 180,E1 -13896.706,E2 -13896.706} C_VEL
LIN {X 0,Y 346.601,Z 377.809,A -85,B 0,C 180,E1 -13897.741,E2 -13897.741} C_VEL
LIN {X 0,Y 346.274,Z 380.391,A -85,B 0,C 180,E1 -13899.535,E2 -13899.535} C_VEL
LIN {X 0,Y 346.042,Z 381.939,A -85,B 0,C 180,E1 -13901.285,E2 -13901.285} C_VEL
LIN {X 0,Y 345.904,Z 382.571,A -85,B 0,C 180,E1 -13903.693,E2 -13903.693} C_VEL
LIN {X 0,Y 345.924,Z 382.028,A -85,B 0,C 180,E1 -13905.322,E2 -13905.322} C_VEL
LIN {X 0,Y 346.04,Z 380.619,A -85,B 0,C 180,E1 -13906.982,E2 -13906.982} C_VEL
LIN {X 0,Y 346.204,Z 378.285,A -85,B 0,C 180,E1 -13908.686,E2 -13908.686} C_VEL
LIN {X 0,Y 346.508,Z 374.93,A -85,B 0,C 180,E1 -13910.419,E2 -13910.419} C_VEL
LIN {X 0,Y 346.867,Z 370.351,A -85,B 0,C 180,E1 -13912.203,E2 -13912.203} C_VEL
LIN {X 0,Y 347.471,Z 364.106,A -85,B 0,C 180,E1 -13914.088,E2 -13914.088} C_VEL
LIN {X 0,Y 348.204,Z 356.702,A -85,B 0,C 180,E1 -13915.844,E2 -13915.844} C_VEL
LIN {X 0,Y 349.067,Z 348.478,A -85,B 0,C 180,E1 -13917.423,E2 -13917.423} C_VEL
LIN {X 0,Y 350.004,Z 338.741,A -85,B 0,C 180,E1 -13918.943,E2 -13918.943} C_VEL
LIN {X 0,Y 351.019,Z 327.836,A -85,B 0,C 180,E1 -13920.296,E2 -13920.296} C_VEL
LIN {X 0,Y 351.975,Z 315.95,A -85,B 0,C 180,E1 -13921.468,E2 -13921.468} C_VEL
LIN {X 0,Y 352.918,Z 303.203,A -85,B 0,C 180,E1 -13922.42,E2 -13922.42} C_VEL
LIN {X 0,Y 353.605,Z 289.776,A -85,B 0,C 180,E1 -13923.153,E2 -13923.153} C_VEL
LIN {X 0,Y 354.119,Z 276.429,A -85,B 0,C 180,E1 -13923.622,E2 -13923.622} C_VEL
LIN {X 0,Y 355.784,Z 198.329,A -85,B 0,C 180,E1 -13925.351,E2 -13925.351} C_VEL
LIN {X 0,Y 351.545,Z 176.316,A -85,B 0,C 180,E1 -13926.1,E2 -13926.1} C_VEL
LIN {X 0,Y 349.981,Z 171.374,A -85,B 0,C 180,E1 -13926.321,E2 -13926.321} C_VEL
LIN {X 0,Y 347.795,Z 160.162,A -85,B 0,C 180,E1 -13929.6,E2 -13929.6} C_VEL
LIN {X 0,Y 347.805,Z 160.163,A -85,B 0,C 180,E1 -13932.357,E2 -13932.357} C_VEL
LIN {X 0,Y 347.894,Z 160.148,A -85,B 0,C 180,E1 -13935.971,E2 -13935.971} C_VEL
LIN {X 0,Y 347.887,Z 160.148,A -85,B 0,C 180,E1 -13939.525,E2 -13939.525} C_VEL
LIN {X 0,Y 348.05,Z 160.127,A -85,B 0,C 180,E1 -13943.042,E2 -13943.042} C_VEL
LIN {X 0,Y 348.184,Z 160.112,A -85,B 0,C 180,E1 -13947.687,E2 -13947.687} C_VEL
LIN {X 0,Y 348.113,Z 160.119,A -85,B 0,C 180,E1 -13951.157,E2 -13951.157} C_VEL
LIN {X 0,Y 348.177,Z 160.114,A -85,B 0,C 180,E1 -13952.314,E2 -13952.314} C_VEL
LIN {X 0,Y 348.049,Z 160.127,A -85,B 0,C 180,E1 -13956.959,E2 -13956.959} C_VEL
LIN {X 0,Y 347.888,Z 160.148,A -85,B 0,C 180,E1 -13960.476,E2 -13960.476} C_VEL
LIN {X 0,Y 347.876,Z 160.151,A -85,B 0,C 180,E1 -13964.137,E2 -13964.137} C_VEL
LIN {X 0,Y 347.789,Z 160.161,A -85,B 0,C 180,E1 -13968.241,E2 -13968.241} C_VEL
LIN {X 0,Y 347.748,Z 160.165,A -85,B 0,C 180,E1 -13970.639,E2 -13970.639} C_VEL
LIN {X 0,Y 347.088,Z 160.253,A -85,B 0,C 180,E1 -13971.605,E2 -13971.605} C_VEL
LIN {X 0,Y 344.232,Z 160.612,A -85,B 0,C 180,E1 -13973.176,E2 -13973.176} C_VEL
LIN {X 0,Y 341.802,Z 160.916,A -85,B 0,C 180,E1 -13974.448,E2 -13974.448} C_VEL
LIN {X 0,Y 340.75,Z 161.043,A -85,B 0,C 180,E1 -13975.433,E2 -13975.433} C_VEL
LIN {X 0,Y 340.661,Z 161.051,A -85,B 0,C 180,E1 -13975.766,E2 -13975.766} C_VEL
LIN {X 0,Y 340.671,Z 161.046,A -85,B 0,C 180,E1 -13978.326,E2 -13978.326} C_VEL
LIN {X 0,Y 340.688,Z 161.047,A -85,B 0,C 180,E1 -13981.045,E2 -13981.045} C_VEL
LIN {X 0,Y 340.713,Z 161.047,A -85,B 0,C 180,E1 -13985.279,E2 -13985.279} C_VEL
LIN {X 0,Y 340.689,Z 161.044,A -85,B 0,C 180,E1 -13988.382,E2 -13988.382} C_VEL
LIN {X 0,Y 340.686,Z 161.045,A -85,B 0,C 180,E1 -13992.044,E2 -13992.044} C_VEL
LIN {X 0,Y 340.645,Z 161.05,A -85,B 0,C 180,E1 -13996.228,E2 -13996.228} C_VEL
LIN {X 0,Y 340.665,Z 161.05,A -85,B 0,C 180,E1 -13998.688,E2 -13998.688} C_VEL
LIN {X 0,Y 340.713,Z 161.041,A -85,B 0,C 180,E1 -14001.771,E2 -14001.771} C_VEL
LIN {X 0,Y 340.717,Z 161.041,A -85,B 0,C 180,E1 -14005.596,E2 -14005.596} C_VEL
LIN {X 0,Y 340.688,Z 161.048,A -85,B 0,C 180,E1 -14008.955,E2 -14008.955} C_VEL
LIN {X 0,Y 340.705,Z 161.045,A -85,B 0,C 180,E1 -14013.012,E2 -14013.012} C_VEL
LIN {X 0,Y 340.695,Z 161.046,A -85,B 0,C 180,E1 -14016.925,E2 -14016.925} C_VEL
LIN {X 0,Y 340.699,Z 161.046,A -85,B 0,C 180,E1 -14020.729,E2 -14020.729} C_VEL
LIN {X 0,Y 340.788,Z 161.037,A -85,B 0,C 180,E1 -14024.45,E2 -14024.45} C_VEL
LIN {X 0,Y 340.839,Z 161.029,A -85,B 0,C 180,E1 -14028.101,E2 -14028.101} C_VEL
LIN {X 0,Y 340.976,Z 161.01,A -85,B 0,C 180,E1 -14031.705,E2 -14031.705} C_VEL
LIN {X 0,Y 341.006,Z 161.009,A -85,B 0,C 180,E1 -14034.086,E2 -14034.086} C_VEL
LIN {X 0,Y 341.113,Z 160.993,A -85,B 0,C 180,E1 -14037.639,E2 -14037.639} C_VEL
LIN {X 0,Y 341.082,Z 160.995,A -85,B 0,C 180,E1 -14041.181,E2 -14041.181} C_VEL
LIN {X 0,Y 341.112,Z 160.994,A -85,B 0,C 180,E1 -14042.362,E2 -14042.362} C_VEL
LIN {X 0,Y 341.006,Z 161.011,A -85,B 0,C 180,E1 -14045.915,E2 -14045.915} C_VEL
LIN {X 0,Y 340.96,Z 161.012,A -85,B 0,C 180,E1 -14048.357,E2 -14048.357} C_VEL
LIN {X 0,Y 340.841,Z 161.03,A -85,B 0,C 180,E1 -14051.9,E2 -14051.9} C_VEL
LIN {X 0,Y 340.785,Z 161.036,A -85,B 0,C 180,E1 -14055.552,E2 -14055.552} C_VEL
LIN {X 0,Y 340.688,Z 161.047,A -85,B 0,C 180,E1 -14059.273,E2 -14059.273} C_VEL
LIN {X 0,Y 340.697,Z 161.045,A -85,B 0,C 180,E1 -14063.076,E2 -14063.076} C_VEL
LIN {X 0,Y 340.707,Z 161.044,A -85,B 0,C 180,E1 -14066.989,E2 -14066.989} C_VEL
LIN {X 0,Y 340.69,Z 161.047,A -85,B 0,C 180,E1 -14071.046,E2 -14071.046} C_VEL
LIN {X 0,Y 340.713,Z 161.047,A -85,B 0,C 180,E1 -14075.28,E2 -14075.28} C_VEL
LIN {X 0,Y 340.691,Z 161.044,A -85,B 0,C 180,E1 -14078.383,E2 -14078.383} C_VEL
LIN {X 0,Y 340.689,Z 161.044,A -85,B 0,C 180,E1 -14082.044,E2 -14082.044} C_VEL
LIN {X 0,Y 340.649,Z 161.049,A -85,B 0,C 180,E1 -14086.228,E2 -14086.228} C_VEL
LIN {X 0,Y 340.668,Z 161.05,A -85,B 0,C 180,E1 -14088.688,E2 -14088.688} C_VEL
LIN {X 0,Y 340.718,Z 161.04,A -85,B 0,C 180,E1 -14091.771,E2 -14091.771} C_VEL
LIN {X 0,Y 340.723,Z 161.04,A -85,B 0,C 180,E1 -14095.596,E2 -14095.596} C_VEL
LIN {X 0,Y 340.697,Z 161.046,A -85,B 0,C 180,E1 -14099.551,E2 -14099.551} C_VEL
LIN {X 0,Y 340.746,Z 161.172,A -85,B 0,C 180,E1 -14099.932,E2 -14099.932} C_VEL
LIN {X 0,Y 343.399,Z 174.262,A -85,B 0,C 180,E1 -14103.512,E2 -14103.512} C_VEL
LIN {X 0,Y 344.398,Z 180.96,A -85,B 0,C 180,E1 -14105.271,E2 -14105.271} C_VEL
LIN {X 0,Y 343.513,Z 189.451,A -85,B 0,C 180,E1 -14107.349,E2 -14107.349} C_VEL
LIN {X 0,Y 348.717,Z 225.629,A -85,B 0,C 180,E1 -14108.511,E2 -14108.511} C_VEL
LIN {X 0,Y 347.061,Z 298.343,A -85,B 0,C 180,E1 -14110.173,E2 -14110.173} C_VEL
LIN {X 0,Y 346.448,Z 311.759,A -85,B 0,C 180,E1 -14110.714,E2 -14110.714} C_VEL
LIN {X 0,Y 345.496,Z 324.562,A -85,B 0,C 180,E1 -14111.468,E2 -14111.468} C_VEL
LIN {X 0,Y 344.457,Z 337.129,A -85,B 0,C 180,E1 -14112.486,E2 -14112.486} C_VEL
LIN {X 0,Y 343.287,Z 348.372,A -85,B 0,C 180,E1 -14113.65,E2 -14113.65} C_VEL
LIN {X 0,Y 342.358,Z 358.652,A -85,B 0,C 180,E1 -14115,E2 -14115} C_VEL
LIN {X 0,Y 341.4,Z 368.523,A -85,B 0,C 180,E1 -14116.609,E2 -14116.609} C_VEL
LIN {X 0,Y 340.426,Z 377.289,A -85,B 0,C 180,E1 -14118.388,E2 -14118.388} C_VEL
LIN {X 0,Y 339.827,Z 384.278,A -85,B 0,C 180,E1 -14120.176,E2 -14120.176} C_VEL
LIN {X 0,Y 339.374,Z 390.681,A -85,B 0,C 180,E1 -14122.264,E2 -14122.264} C_VEL
LIN {X 0,Y 339.172,Z 394.839,A -85,B 0,C 180,E1 -14124.053,E2 -14124.053} C_VEL
LIN {X 0,Y 339.073,Z 396.992,A -85,B 0,C 180,E1 -14125.244,E2 -14125.244} C_VEL
LIN {X 0,Y 339.071,Z 398.681,A -85,B 0,C 180,E1 -14126.435,E2 -14126.435} C_VEL
LIN {X 0,Y 339.001,Z 399.951,A -85,B 0,C 180,E1 -14127.624,E2 -14127.624} C_VEL
LIN {X 0,Y 339.021,Z 400.808,A -85,B 0,C 180,E1 -14128.812,E2 -14128.812} C_VEL
LIN {X 0,Y 339.069,Z 401.212,A -85,B 0,C 180,E1 -14130,E2 -14130} C_VEL
LIN {X 0,Y 339.007,Z 401.209,A -85,B 0,C 180,E1 -14131.188,E2 -14131.188} C_VEL
LIN {X 0,Y 338.997,Z 400.812,A -85,B 0,C 180,E1 -14132.376,E2 -14132.376} C_VEL
LIN {X 0,Y 339.065,Z 400.01,A -85,B 0,C 180,E1 -14133.565,E2 -14133.565} C_VEL
LIN {X 0,Y 339.112,Z 397.236,A -85,B 0,C 180,E1 -14135.849,E2 -14135.849} C_VEL
LIN {X 0,Y 339.404,Z 393.744,A -85,B 0,C 180,E1 -14137.735,E2 -14137.735} C_VEL
LIN {X 0,Y 339.851,Z 389.334,A -85,B 0,C 180,E1 -14139.522,E2 -14139.522} C_VEL
LIN {X 0,Y 340.591,Z 383.73,A -85,B 0,C 180,E1 -14141.305,E2 -14141.305} C_VEL
LIN {X 0,Y 341.52,Z 376.752,A -85,B 0,C 180,E1 -14143.083,E2 -14143.083} C_VEL
LIN {X 0,Y 342.841,Z 368.046,A -85,B 0,C 180,E1 -14144.847,E2 -14144.847} C_VEL
LIN {X 0,Y 343.91,Z 359.163,A -85,B 0,C 180,E1 -14146.317,E2 -14146.317} C_VEL
LIN {X 0,Y 345.403,Z 348.236,A -85,B 0,C 180,E1 -14147.77,E2 -14147.77} C_VEL
LIN {X 0,Y 346.856,Z 337.271,A -85,B 0,C 180,E1 -14148.916,E2 -14148.916} C_VEL
LIN {X 0,Y 348.143,Z 325.096,A -85,B 0,C 180,E1 -14149.916,E2 -14149.916} C_VEL
LIN {X 0,Y 349.325,Z 312.427,A -85,B 0,C 180,E1 -14150.691,E2 -14150.691} C_VEL
LIN {X 0,Y 350.233,Z 299.039,A -85,B 0,C 180,E1 -14151.25,E2 -14151.25} C_VEL
LIN {X 0,Y 351.03,Z 276.189,A -85,B 0,C 180,E1 -14151.816,E2 -14151.816} C_VEL
LIN {X 0,Y 352.317,Z 225.065,A -85,B 0,C 180,E1 -14153.012,E2 -14153.012} C_VEL
LIN {X 0,Y 349.002,Z 204.831,A -85,B 0,C 180,E1 -14153.824,E2 -14153.824} C_VEL
LIN {X 0,Y 345.423,Z 187.752,A -85,B 0,C 180,E1 -14154.636,E2 -14154.636} C_VEL
LIN {X 0,Y 345.707,Z 184.128,A -85,B 0,C 180,E1 -14155.548,E2 -14155.548} C_VEL
LIN {X 0,Y 343.772,Z 173.784,A -85,B 0,C 180,E1 -14158.467,E2 -14158.467} C_VEL
LIN {X 0,Y 341.536,Z 164.389,A -85,B 0,C 180,E1 -14161.304,E2 -14161.304} C_VEL
LIN {X 0,Y 340.691,Z 161.052,A -85,B 0,C 180,E1 -14162.358,E2 -14162.358} C_VEL
LIN {X 0,Y 340.714,Z 161.045,A -85,B 0,C 180,E1 -14165.278,E2 -14165.278} C_VEL
LIN {X 0,Y 340.691,Z 161.049,A -85,B 0,C 180,E1 -14168.381,E2 -14168.381} C_VEL
LIN {X 0,Y 340.688,Z 161.051,A -85,B 0,C 180,E1 -14172.043,E2 -14172.043} C_VEL
LIN {X 0,Y 340.647,Z 161.054,A -85,B 0,C 180,E1 -14176.227,E2 -14176.227} C_VEL
LIN {X 0,Y 340.666,Z 161.051,A -85,B 0,C 180,E1 -14178.687,E2 -14178.687} C_VEL
LIN {X 0,Y 340.715,Z 161.044,A -85,B 0,C 180,E1 -14181.77,E2 -14181.77} C_VEL
LIN {X 0,Y 340.718,Z 161.041,A -85,B 0,C 180,E1 -14185.595,E2 -14185.595} C_VEL
LIN {X 0,Y 340.688,Z 161.044,A -85,B 0,C 180,E1 -14188.954,E2 -14188.954} C_VEL
LIN {X 0,Y 340.705,Z 161.038,A -85,B 0,C 180,E1 -14193.011,E2 -14193.011} C_VEL
LIN {X 0,Y 340.695,Z 161.038,A -85,B 0,C 180,E1 -14196.924,E2 -14196.924} C_VEL
LIN {X 0,Y 340.692,Z 161.039,A -85,B 0,C 180,E1 -14200.727,E2 -14200.727} C_VEL
LIN {X 0,Y 340.782,Z 161.029,A -85,B 0,C 180,E1 -14204.448,E2 -14204.448} C_VEL
LIN {X 0,Y 340.838,Z 161.023,A -85,B 0,C 180,E1 -14208.1,E2 -14208.1} C_VEL
LIN {X 0,Y 340.974,Z 161.006,A -85,B 0,C 180,E1 -14211.704,E2 -14211.704} C_VEL
LIN {X 0,Y 341.004,Z 161.007,A -85,B 0,C 180,E1 -14214.085,E2 -14214.085} C_VEL
LIN {X 0,Y 341.117,Z 160.992,A -85,B 0,C 180,E1 -14217.638,E2 -14217.638} C_VEL
LIN {X 0,Y 341.08,Z 160.994,A -85,B 0,C 180,E1 -14221.18,E2 -14221.18} C_VEL
LIN {X 0,Y 341.116,Z 160.995,A -85,B 0,C 180,E1 -14222.361,E2 -14222.361} C_VEL
LIN {X 0,Y 340.992,Z 161.011,A -85,B 0,C 180,E1 -14227.103,E2 -14227.103} C_VEL
LIN {X 0,Y 340.836,Z 161.034,A -85,B 0,C 180,E1 -14230.694,E2 -14230.694} C_VEL
LIN {X 0,Y 340.812,Z 161.039,A -85,B 0,C 180,E1 -14234.327,E2 -14234.327} C_VEL
LIN {X 0,Y 340.775,Z 161.155,A -85,B 0,C 180,E1 -14235.666,E2 -14235.666} C_VEL
LIN {X 0,Y 342.944,Z 170.115,A -85,B 0,C 180,E1 -14238.52,E2 -14238.52} C_VEL
LIN {X 0,Y 343.553,Z 172.77,A -85,B 0,C 180,E1 -14239.274,E2 -14239.274} C_VEL
LIN {X 0,Y 350.049,Z 187.806,A -85,B 0,C 180,E1 -14240.289,E2 -14240.289} C_VEL
LIN {X 0,Y 352.953,Z 201.11,A -85,B 0,C 180,E1 -14240.888,E2 -14240.888} C_VEL
LIN {X 0,Y 350.595,Z 280.804,A -85,B 0,C 180,E1 -14242.766,E2 -14242.766} C_VEL
LIN {X 0,Y 349.857,Z 293.905,A -85,B 0,C 180,E1 -14243.301,E2 -14243.301} C_VEL
LIN {X 0,Y 348.952,Z 306.328,A -85,B 0,C 180,E1 -14244.042,E2 -14244.042} C_VEL
LIN {X 0,Y 347.797,Z 318.129,A -85,B 0,C 180,E1 -14244.988,E2 -14244.988} C_VEL
LIN {X 0,Y 346.479,Z 329.701,A -85,B 0,C 180,E1 -14246.179,E2 -14246.179} C_VEL
LIN {X 0,Y 345.113,Z 339.512,A -85,B 0,C 180,E1 -14247.434,E2 -14247.434} C_VEL
LIN {X 0,Y 343.847,Z 348.915,A -85,B 0,C 180,E1 -14248.939,E2 -14248.939} C_VEL
LIN {X 0,Y 342.628,Z 356.949,A -85,B 0,C 180,E1 -14250.516,E2 -14250.516} C_VEL
LIN {X 0,Y 341.487,Z 364.484,A -85,B 0,C 180,E1 -14252.35,E2 -14252.35} C_VEL
LIN {X 0,Y 340.55,Z 370.929,A -85,B 0,C 180,E1 -14254.364,E2 -14254.364} C_VEL
LIN {X 0,Y 339.896,Z 375.553,A -85,B 0,C 180,E1 -14256.256,E2 -14256.256} C_VEL
LIN {X 0,Y 339.362,Z 379.357,A -85,B 0,C 180,E1 -14258.409,E2 -14258.409} C_VEL
LIN {X 0,Y 339.122,Z 381.208,A -85,B 0,C 180,E1 -14259.974,E2 -14259.974} C_VEL
LIN {X 0,Y 338.916,Z 382.435,A -85,B 0,C 180,E1 -14261.711,E2 -14261.711} C_VEL
LIN {X 0,Y 338.81,Z 382.797,A -85,B 0,C 180,E1 -14263.448,E2 -14263.448} C_VEL
LIN {X 0,Y 338.829,Z 382.291,A -85,B 0,C 180,E1 -14265.153,E2 -14265.153} C_VEL
LIN {X 0,Y 338.946,Z 380.962,A -85,B 0,C 180,E1 -14266.824,E2 -14266.824} C_VEL
LIN {X 0,Y 339.088,Z 378.878,A -85,B 0,C 180,E1 -14268.454,E2 -14268.454} C_VEL
LIN {X 0,Y 339.335,Z 376.028,A -85,B 0,C 180,E1 -14270.057,E2 -14270.057} C_VEL
LIN {X 0,Y 339.704,Z 371.85,A -85,B 0,C 180,E1 -14271.828,E2 -14271.828} C_VEL
LIN {X 0,Y 340.23,Z 366.241,A -85,B 0,C 180,E1 -14273.668,E2 -14273.668} C_VEL
LIN {X 0,Y 340.939,Z 359.014,A -85,B 0,C 180,E1 -14275.541,E2 -14275.541} C_VEL
LIN {X 0,Y 341.762,Z 351.131,A -85,B 0,C 180,E1 -14277.183,E2 -14277.183} C_VEL
LIN {X 0,Y 342.811,Z 341.273,A -85,B 0,C 180,E1 -14278.826,E2 -14278.826} C_VEL
LIN {X 0,Y 343.908,Z 330.292,A -85,B 0,C 180,E1 -14280.294,E2 -14280.294} C_VEL
LIN {X 0,Y 344.876,Z 319.023,A -85,B 0,C 180,E1 -14281.481,E2 -14281.481} C_VEL
LIN {X 0,Y 345.833,Z 306.924,A -85,B 0,C 180,E1 -14282.475,E2 -14282.475} C_VEL
LIN {X 0,Y 346.553,Z 295.199,A -85,B 0,C 180,E1 -14283.206,E2 -14283.206} C_VEL
LIN {X 0,Y 347.09,Z 282.264,A -85,B 0,C 180,E1 -14283.77,E2 -14283.77} C_VEL
LIN {X 0,Y 347.591,Z 263.19,A -85,B 0,C 180,E1 -14284.254,E2 -14284.254} C_VEL
LIN {X 0,Y 348.974,Z 198.775,A -85,B 0,C 180,E1 -14285.706,E2 -14285.706} C_VEL
LIN {X 0,Y 345.095,Z 178.603,A -85,B 0,C 180,E1 -14286.41,E2 -14286.41} C_VEL
LIN {X 0,Y 342.772,Z 171.493,A -85,B 0,C 180,E1 -14286.75,E2 -14286.75} C_VEL
LIN {X 0,Y 340.748,Z 161.039,A -85,B 0,C 180,E1 -14289.869,E2 -14289.869} C_VEL
LIN {X 0,Y 340.736,Z 161.038,A -85,B 0,C 180,E1 -14293.217,E2 -14293.217} C_VEL
LIN {X 0,Y 340.837,Z 161.027,A -85,B 0,C 180,E1 -14296.891,E2 -14296.891} C_VEL
LIN {X 0,Y 340.876,Z 161.025,A -85,B 0,C 180,E1 -14300.507,E2 -14300.507} C_VEL
LIN {X 0,Y 340.998,Z 161.006,A -85,B 0,C 180,E1 -14302.897,E2 -14302.897} C_VEL
LIN {X 0,Y 340.806,Z 161.029,A -85,B 0,C 180,E1 -14305.269,E2 -14305.269} C_VEL
LIN {X 0,Y 341.121,Z 160.992,A -85,B 0,C 180,E1 -14307.639,E2 -14307.639} C_VEL
LIN {X 0,Y 341.084,Z 160.995,A -85,B 0,C 180,E1 -14311.181,E2 -14311.181} C_VEL
LIN {X 0,Y 341.114,Z 160.994,A -85,B 0,C 180,E1 -14312.362,E2 -14312.362} C_VEL
LIN {X 0,Y 341.008,Z 161.01,A -85,B 0,C 180,E1 -14315.915,E2 -14315.915} C_VEL
LIN {X 0,Y 340.96,Z 161.012,A -85,B 0,C 180,E1 -14318.356,E2 -14318.356} C_VEL
LIN {X 0,Y 340.842,Z 161.03,A -85,B 0,C 180,E1 -14321.9,E2 -14321.9} C_VEL
LIN {X 0,Y 340.785,Z 161.036,A -85,B 0,C 180,E1 -14325.551,E2 -14325.551} C_VEL
LIN {X 0,Y 340.696,Z 161.045,A -85,B 0,C 180,E1 -14329.272,E2 -14329.272} C_VEL
LIN {X 0,Y 340.696,Z 161.045,A -85,B 0,C 180,E1 -14333.075,E2 -14333.075} C_VEL
LIN {X 0,Y 340.661,Z 161.051,A -85,B 0,C 180,E1 -14335.766,E2 -14335.766} C_VEL
LIN {X 0,Y 339.986,Z 161.133,A -85,B 0,C 180,E1 -14336.753,E2 -14336.753} C_VEL
LIN {X 0,Y 337.147,Z 161.485,A -85,B 0,C 180,E1 -14338.359,E2 -14338.359} C_VEL
LIN {X 0,Y 334.742,Z 161.788,A -85,B 0,C 180,E1 -14339.66,E2 -14339.66} C_VEL
LIN {X 0,Y 333.703,Z 161.915,A -85,B 0,C 180,E1 -14340.666,E2 -14340.666} C_VEL
LIN {X 0,Y 333.615,Z 161.923,A -85,B 0,C 180,E1 -14341.007,E2 -14341.007} C_VEL
LIN {X 0,Y 333.681,Z 161.918,A -85,B 0,C 180,E1 -14344.774,E2 -14344.774} C_VEL
LIN {X 0,Y 333.639,Z 161.924,A -85,B 0,C 180,E1 -14347.652,E2 -14347.652} C_VEL
LIN {X 0,Y 333.598,Z 161.93,A -85,B 0,C 180,E1 -14350.774,E2 -14350.774} C_VEL
LIN {X 0,Y 333.585,Z 161.929,A -85,B 0,C 180,E1 -14354.25,E2 -14354.25} C_VEL
LIN {X 0,Y 333.631,Z 161.924,A -85,B 0,C 180,E1 -14357.618,E2 -14357.618} C_VEL
LIN {X 0,Y 333.629,Z 161.927,A -85,B 0,C 180,E1 -14361.206,E2 -14361.206} C_VEL
LIN {X 0,Y 333.668,Z 161.919,A -85,B 0,C 180,E1 -14363.861,E2 -14363.861} C_VEL
LIN {X 0,Y 333.639,Z 161.923,A -85,B 0,C 180,E1 -14367.413,E2 -14367.413} C_VEL
LIN {X 0,Y 333.646,Z 161.924,A -85,B 0,C 180,E1 -14371.022,E2 -14371.022} C_VEL
LIN {X 0,Y 333.658,Z 161.922,A -85,B 0,C 180,E1 -14375.086,E2 -14375.086} C_VEL
LIN {X 0,Y 333.647,Z 161.923,A -85,B 0,C 180,E1 -14379.018,E2 -14379.018} C_VEL
LIN {X 0,Y 333.707,Z 161.914,A -85,B 0,C 180,E1 -14381.585,E2 -14381.585} C_VEL
LIN {X 0,Y 333.769,Z 161.906,A -85,B 0,C 180,E1 -14385.601,E2 -14385.601} C_VEL
LIN {X 0,Y 333.808,Z 161.902,A -85,B 0,C 180,E1 -14389.078,E2 -14389.078} C_VEL
LIN {X 0,Y 333.95,Z 161.885,A -85,B 0,C 180,E1 -14392.746,E2 -14392.746} C_VEL
LIN {X 0,Y 333.769,Z 161.906,A -85,B 0,C 180,E1 -14395.169,E2 -14395.169} C_VEL
LIN {X 0,Y 334.053,Z 161.872,A -85,B 0,C 180,E1 -14397.589,E2 -14397.589} C_VEL
LIN {X 0,Y 334.053,Z 161.871,A -85,B 0,C 180,E1 -14401.206,E2 -14401.206} C_VEL
LIN {X 0,Y 334.053,Z 161.873,A -85,B 0,C 180,E1 -14402.412,E2 -14402.412} C_VEL
LIN {X 0,Y 333.98,Z 161.885,A -85,B 0,C 180,E1 -14406.04,E2 -14406.04} C_VEL
LIN {X 0,Y 333.91,Z 161.89,A -85,B 0,C 180,E1 -14408.473,E2 -14408.473} C_VEL
LIN {X 0,Y 333.782,Z 161.907,A -85,B 0,C 180,E1 -14412.155,E2 -14412.155} C_VEL
LIN {X 0,Y 333.748,Z 161.909,A -85,B 0,C 180,E1 -14414.637,E2 -14414.637} C_VEL
LIN {X 0,Y 333.69,Z 161.916,A -85,B 0,C 180,E1 -14418.602,E2 -14418.602} C_VEL
LIN {X 0,Y 333.646,Z 161.922,A -85,B 0,C 180,E1 -14422.282,E2 -14422.282} C_VEL
LIN {X 0,Y 333.653,Z 161.923,A -85,B 0,C 180,E1 -14425.078,E2 -14425.078} C_VEL
LIN {X 0,Y 333.626,Z 161.926,A -85,B 0,C 180,E1 -14428.981,E2 -14428.981} C_VEL
LIN {X 0,Y 333.642,Z 161.922,A -85,B 0,C 180,E1 -14432.587,E2 -14432.587} C_VEL
LIN {X 0,Y 333.671,Z 161.918,A -85,B 0,C 180,E1 -14436.14,E2 -14436.14} C_VEL
LIN {X 0,Y 333.618,Z 161.931,A -85,B 0,C 180,E1 -14439.197,E2 -14439.197} C_VEL
LIN {X 0,Y 333.625,Z 161.925,A -85,B 0,C 180,E1 -14442.499,E2 -14442.499} C_VEL
LIN {X 0,Y 333.593,Z 161.928,A -85,B 0,C 180,E1 -14445.955,E2 -14445.955} C_VEL
LIN {X 0,Y 333.601,Z 161.929,A -85,B 0,C 180,E1 -14449.325,E2 -14449.325} C_VEL
LIN {X 0,Y 333.661,Z 161.922,A -85,B 0,C 180,E1 -14453.169,E2 -14453.169} C_VEL
LIN {X 0,Y 333.673,Z 161.919,A -85,B 0,C 180,E1 -14455.342,E2 -14455.342} C_VEL
LIN {X 0,Y 333.685,Z 161.956,A -85,B 0,C 180,E1 -14459.593,E2 -14459.593} C_VEL
LIN {X 0,Y 336.397,Z 175.218,A -85,B 0,C 180,E1 -14463.308,E2 -14463.308} C_VEL
LIN {X 0,Y 337.419,Z 181.709,A -85,B 0,C 180,E1 -14465.053,E2 -14465.053} C_VEL
LIN {X 0,Y 336.607,Z 189.27,A -85,B 0,C 180,E1 -14466.941,E2 -14466.941} C_VEL
LIN {X 0,Y 341.958,Z 225.802,A -85,B 0,C 180,E1 -14468.151,E2 -14468.151} C_VEL
LIN {X 0,Y 340.261,Z 298.055,A -85,B 0,C 180,E1 -14469.838,E2 -14469.838} C_VEL
LIN {X 0,Y 339.63,Z 311.489,A -85,B 0,C 180,E1 -14470.39,E2 -14470.39} C_VEL
LIN {X 0,Y 338.642,Z 324.314,A -85,B 0,C 180,E1 -14471.157,E2 -14471.157} C_VEL
LIN {X 0,Y 337.615,Z 336.093,A -85,B 0,C 180,E1 -14472.119,E2 -14472.119} C_VEL
LIN {X 0,Y 336.407,Z 347.49,A -85,B 0,C 180,E1 -14473.306,E2 -14473.306} C_VEL
LIN {X 0,Y 335.488,Z 357.741,A -85,B 0,C 180,E1 -14474.654,E2 -14474.654} C_VEL
LIN {X 0,Y 334.424,Z 367.898,A -85,B 0,C 180,E1 -14476.325,E2 -14476.325} C_VEL
LIN {X 0,Y 333.419,Z 376.766,A -85,B 0,C 180,E1 -14478.14,E2 -14478.14} C_VEL
LIN {X 0,Y 332.789,Z 383.823,A -85,B 0,C 180,E1 -14479.966,E2 -14479.966} C_VEL
LIN {X 0,Y 332.31,Z 390.281,A -85,B 0,C 180,E1 -14482.099,E2 -14482.099} C_VEL
LIN {X 0,Y 332.081,Z 394.835,A -85,B 0,C 180,E1 -14484.094,E2 -14484.094} C_VEL
LIN {X 0,Y 331.996,Z 398.397,A -85,B 0,C 180,E1 -14486.359,E2 -14486.359} C_VEL
LIN {X 0,Y 331.918,Z 399.687,A -85,B 0,C 180,E1 -14487.573,E2 -14487.573} C_VEL
LIN {X 0,Y 331.926,Z 400.571,A -85,B 0,C 180,E1 -14488.787,E2 -14488.787} C_VEL
LIN {X 0,Y 331.971,Z 401.005,A -85,B 0,C 180,E1 -14490,E2 -14490} C_VEL
LIN {X 0,Y 331.913,Z 401.021,A -85,B 0,C 180,E1 -14491.213,E2 -14491.213} C_VEL
LIN {X 0,Y 331.914,Z 400.642,A -85,B 0,C 180,E1 -14492.427,E2 -14492.427} C_VEL
LIN {X 0,Y 331.968,Z 399.867,A -85,B 0,C 180,E1 -14493.641,E2 -14493.641} C_VEL
LIN {X 0,Y 332.007,Z 397.444,A -85,B 0,C 180,E1 -14495.78,E2 -14495.78} C_VEL
LIN {X 0,Y 332.361,Z 393.706,A -85,B 0,C 180,E1 -14497.9,E2 -14497.9} C_VEL
LIN {X 0,Y 332.821,Z 389.342,A -85,B 0,C 180,E1 -14499.725,E2 -14499.725} C_VEL
LIN {X 0,Y 333.702,Z 382.755,A -85,B 0,C 180,E1 -14501.849,E2 -14501.849} C_VEL
LIN {X 0,Y 334.85,Z 375.552,A -85,B 0,C 180,E1 -14503.657,E2 -14503.657} C_VEL
LIN {X 0,Y 336.181,Z 366.598,A -85,B 0,C 180,E1 -14505.458,E2 -14505.458} C_VEL
LIN {X 0,Y 337.409,Z 357.453,A -85,B 0,C 180,E1 -14506.954,E2 -14506.954} C_VEL
LIN {X 0,Y 338.844,Z 347.423,A -85,B 0,C 180,E1 -14508.282,E2 -14508.282} C_VEL
LIN {X 0,Y 340.358,Z 336.337,A -85,B 0,C 180,E1 -14509.448,E2 -14509.448} C_VEL
LIN {X 0,Y 341.758,Z 324.03,A -85,B 0,C 180,E1 -14510.462,E2 -14510.462} C_VEL
LIN {X 0,Y 342.948,Z 311.022,A -85,B 0,C 180,E1 -14511.251,E2 -14511.251} C_VEL
LIN {X 0,Y 343.907,Z 297.103,A -85,B 0,C 180,E1 -14511.818,E2 -14511.818} C_VEL
LIN {X 0,Y 345.991,Z 225.915,A -85,B 0,C 180,E1 -14513.532,E2 -14513.532} C_VEL
LIN {X 0,Y 342.904,Z 206.851,A -85,B 0,C 180,E1 -14514.321,E2 -14514.321} C_VEL
LIN {X 0,Y 338.818,Z 187.536,A -85,B 0,C 180,E1 -14515.278,E2 -14515.278} C_VEL
LIN {X 0,Y 338.674,Z 184.345,A -85,B 0,C 180,E1 -14516.139,E2 -14516.139} C_VEL
LIN {X 0,Y 336.462,Z 173.251,A -85,B 0,C 180,E1 -14519.396,E2 -14519.396} C_VEL
LIN {X 0,Y 334.297,Z 164.508,A -85,B 0,C 180,E1 -14522.15,E2 -14522.15} C_VEL
LIN {X 0,Y 333.629,Z 161.93,A -85,B 0,C 180,E1 -14523.025,E2 -14523.025} C_VEL
LIN {X 0,Y 333.672,Z 161.923,A -85,B 0,C 180,E1 -14526.139,E2 -14526.139} C_VEL
LIN {X 0,Y 333.618,Z 161.933,A -85,B 0,C 180,E1 -14529.195,E2 -14529.195} C_VEL
LIN {X 0,Y 333.624,Z 161.929,A -85,B 0,C 180,E1 -14532.498,E2 -14532.498} C_VEL
LIN {X 0,Y 333.59,Z 161.933,A -85,B 0,C 180,E1 -14535.953,E2 -14535.953} C_VEL
LIN {X 0,Y 333.599,Z 161.93,A -85,B 0,C 180,E1 -14539.324,E2 -14539.324} C_VEL
LIN {X 0,Y 333.658,Z 161.917,A -85,B 0,C 180,E1 -14543.168,E2 -14543.168} C_VEL
LIN {X 0,Y 333.669,Z 161.92,A -85,B 0,C 180,E1 -14545.34,E2 -14545.34} C_VEL
LIN {X 0,Y 333.625,Z 161.926,A -85,B 0,C 180,E1 -14548.221,E2 -14548.221} C_VEL
LIN {X 0,Y 333.644,Z 161.922,A -85,B 0,C 180,E1 -14551.021,E2 -14551.021} C_VEL
LIN {X 0,Y 333.658,Z 161.923,A -85,B 0,C 180,E1 -14555.085,E2 -14555.085} C_VEL
LIN {X 0,Y 333.644,Z 161.925,A -85,B 0,C 180,E1 -14559.016,E2 -14559.016} C_VEL
LIN {X 0,Y 333.7,Z 161.91,A -85,B 0,C 180,E1 -14561.584,E2 -14561.584} C_VEL
LIN {X 0,Y 333.768,Z 161.904,A -85,B 0,C 180,E1 -14565.6,E2 -14565.6} C_VEL
LIN {X 0,Y 333.807,Z 161.901,A -85,B 0,C 180,E1 -14569.077,E2 -14569.077} C_VEL
LIN {X 0,Y 333.948,Z 161.886,A -85,B 0,C 180,E1 -14572.745,E2 -14572.745} C_VEL
LIN {X 0,Y 333.767,Z 161.902,A -85,B 0,C 180,E1 -14575.168,E2 -14575.168} C_VEL
LIN {X 0,Y 334.057,Z 161.872,A -85,B 0,C 180,E1 -14577.588,E2 -14577.588} C_VEL
LIN {X 0,Y 334.051,Z 161.87,A -85,B 0,C 180,E1 -14581.205,E2 -14581.205} C_VEL
LIN {X 0,Y 334.057,Z 161.874,A -85,B 0,C 180,E1 -14582.411,E2 -14582.411} C_VEL
LIN {X 0,Y 333.95,Z 161.884,A -85,B 0,C 180,E1 -14586.462,E2 -14586.462} C_VEL
LIN {X 0,Y 333.811,Z 161.907,A -85,B 0,C 180,E1 -14589.696,E2 -14589.696} C_VEL
LIN {X 0,Y 333.776,Z 161.917,A -85,B 0,C 180,E1 -14593.392,E2 -14593.392} C_VEL
LIN {X 0,Y 333.755,Z 162.016,A -85,B 0,C 180,E1 -14595.026,E2 -14595.026} C_VEL
LIN {X 0,Y 336.253,Z 172.379,A -85,B 0,C 180,E1 -14598.428,E2 -14598.428} C_VEL
LIN {X 0,Y 336.455,Z 173.127,A -85,B 0,C 180,E1 -14598.575,E2 -14598.575} C_VEL
LIN {X 0,Y 343.356,Z 188.549,A -85,B 0,C 180,E1 -14599.689,E2 -14599.689} C_VEL
LIN {X 0,Y 344.848,Z 193.234,A -85,B 0,C 180,E1 -14599.96,E2 -14599.96} C_VEL
LIN {X 0,Y 346.701,Z 203.213,A -85,B 0,C 180,E1 -14600.395,E2 -14600.395} C_VEL
LIN {X 0,Y 344.202,Z 281.357,A -85,B 0,C 180,E1 -14602.272,E2 -14602.272} C_VEL
LIN {X 0,Y 343.364,Z 294.966,A -85,B 0,C 180,E1 -14602.845,E2 -14602.845} C_VEL
LIN {X 0,Y 342.399,Z 307.357,A -85,B 0,C 180,E1 -14603.617,E2 -14603.617} C_VEL
LIN {X 0,Y 341.18,Z 319.077,A -85,B 0,C 180,E1 -14604.59,E2 -14604.59} C_VEL
LIN {X 0,Y 339.859,Z 329.937,A -85,B 0,C 180,E1 -14605.738,E2 -14605.738} C_VEL
LIN {X 0,Y 338.487,Z 339.269,A -85,B 0,C 180,E1 -14606.952,E2 -14606.952} C_VEL
LIN {X 0,Y 337.166,Z 348.703,A -85,B 0,C 180,E1 -14608.477,E2 -14608.477} C_VEL
LIN {X 0,Y 335.835,Z 357.101,A -85,B 0,C 180,E1 -14610.148,E2 -14610.148} C_VEL
LIN {X 0,Y 334.658,Z 364.309,A -85,B 0,C 180,E1 -14611.925,E2 -14611.925} C_VEL
LIN {X 0,Y 333.667,Z 370.727,A -85,B 0,C 180,E1 -14613.928,E2 -14613.928} C_VEL
LIN {X 0,Y 332.826,Z 376.233,A -85,B 0,C 180,E1 -14616.245,E2 -14616.245} C_VEL
LIN {X 0,Y 332.252,Z 379.969,A -85,B 0,C 180,E1 -14618.498,E2 -14618.498} C_VEL
LIN {X 0,Y 331.972,Z 381.899,A -85,B 0,C 180,E1 -14620.348,E2 -14620.348} C_VEL
LIN {X 0,Y 331.717,Z 382.948,A -85,B 0,C 180,E1 -14622.685,E2 -14622.685} C_VEL
LIN {X 0,Y 331.717,Z 382.807,A -85,B 0,C 180,E1 -14624.359,E2 -14624.359} C_VEL
LIN {X 0,Y 331.776,Z 381.845,A -85,B 0,C 180,E1 -14626.072,E2 -14626.072} C_VEL
LIN {X 0,Y 331.931,Z 379.995,A -85,B 0,C 180,E1 -14627.821,E2 -14627.821} C_VEL
LIN {X 0,Y 332.14,Z 377.166,A -85,B 0,C 180,E1 -14629.618,E2 -14629.618} C_VEL
LIN {X 0,Y 332.619,Z 372.276,A -85,B 0,C 180,E1 -14631.833,E2 -14631.833} C_VEL
LIN {X 0,Y 333.177,Z 366.424,A -85,B 0,C 180,E1 -14633.799,E2 -14633.799} C_VEL
LIN {X 0,Y 333.954,Z 359.067,A -85,B 0,C 180,E1 -14635.741,E2 -14635.741} C_VEL
LIN {X 0,Y 334.777,Z 351.234,A -85,B 0,C 180,E1 -14637.4,E2 -14637.4} C_VEL
LIN {X 0,Y 335.859,Z 341.289,A -85,B 0,C 180,E1 -14639.085,E2 -14639.085} C_VEL
LIN {X 0,Y 336.966,Z 330.728,A -85,B 0,C 180,E1 -14640.525,E2 -14640.525} C_VEL
LIN {X 0,Y 338.005,Z 319.171,A -85,B 0,C 180,E1 -14641.769,E2 -14641.769} C_VEL
LIN {X 0,Y 338.999,Z 307.074,A -85,B 0,C 180,E1 -14642.782,E2 -14642.782} C_VEL
LIN {X 0,Y 339.729,Z 295.642,A -85,B 0,C 180,E1 -14643.509,E2 -14643.509} C_VEL
LIN {X 0,Y 340.28,Z 282.711,A -85,B 0,C 180,E1 -14644.091,E2 -14644.091} C_VEL
LIN {X 0,Y 340.755,Z 264.913,A -85,B 0,C 180,E1 -14644.561,E2 -14644.561} C_VEL
LIN {X 0,Y 342.311,Z 200.188,A -85,B 0,C 180,E1 -14646.043,E2 -14646.043} C_VEL
LIN {X 0,Y 338.616,Z 180.843,A -85,B 0,C 180,E1 -14646.735,E2 -14646.735} C_VEL
LIN {X 0,Y 335.612,Z 171.769,A -85,B 0,C 180,E1 -14647.151,E2 -14647.151} C_VEL
LIN {X 0,Y 333.682,Z 161.92,A -85,B 0,C 180,E1 -14650.147,E2 -14650.147} C_VEL
LIN {X 0,Y 333.713,Z 161.916,A -85,B 0,C 180,E1 -14654.111,E2 -14654.111} C_VEL
LIN {X 0,Y 333.783,Z 161.906,A -85,B 0,C 180,E1 -14657.845,E2 -14657.845} C_VEL
LIN {X 0,Y 333.92,Z 161.888,A -85,B 0,C 180,E1 -14661.57,E2 -14661.57} C_VEL
LIN {X 0,Y 333.984,Z 161.883,A -85,B 0,C 180,E1 -14663.961,E2 -14663.961} C_VEL
LIN {X 0,Y 334.061,Z 161.871,A -85,B 0,C 180,E1 -14667.589,E2 -14667.589} C_VEL
LIN {X 0,Y 334.054,Z 161.871,A -85,B 0,C 180,E1 -14671.206,E2 -14671.206} C_VEL
LIN {X 0,Y 334.055,Z 161.873,A -85,B 0,C 180,E1 -14672.412,E2 -14672.412} C_VEL
LIN {X 0,Y 333.982,Z 161.885,A -85,B 0,C 180,E1 -14676.04,E2 -14676.04} C_VEL
LIN {X 0,Y 333.91,Z 161.89,A -85,B 0,C 180,E1 -14678.472,E2 -14678.472} C_VEL
LIN {X 0,Y 333.783,Z 161.907,A -85,B 0,C 180,E1 -14682.155,E2 -14682.155} C_VEL
LIN {X 0,Y 333.748,Z 161.909,A -85,B 0,C 180,E1 -14684.637,E2 -14684.637} C_VEL
LIN {X 0,Y 333.69,Z 161.916,A -85,B 0,C 180,E1 -14688.602,E2 -14688.602} C_VEL
LIN {X 0,Y 333.645,Z 161.922,A -85,B 0,C 180,E1 -14692.281,E2 -14692.281} C_VEL
LIN {X 0,Y 333.618,Z 161.924,A -85,B 0,C 180,E1 -14695.763,E2 -14695.763} C_VEL
LIN {X 0,Y 333.624,Z 161.926,A -85,B 0,C 180,E1 -14698.98,E2 -14698.98} C_VEL
LIN {X 0,Y 333.615,Z 161.923,A -85,B 0,C 180,E1 -14701.007,E2 -14701.007} C_VEL
LIN {X 0,Y 332.935,Z 162.012,A -85,B 0,C 180,E1 -14702.014,E2 -14702.014} C_VEL
LIN {X 0,Y 330.081,Z 162.368,A -85,B 0,C 180,E1 -14703.654,E2 -14703.654} C_VEL
LIN {X 0,Y 327.679,Z 162.667,A -85,B 0,C 180,E1 -14704.983,E2 -14704.983} C_VEL
LIN {X 0,Y 326.662,Z 162.792,A -85,B 0,C 180,E1 -14706.011,E2 -14706.011} C_VEL
LIN {X 0,Y 326.587,Z 162.801,A -85,B 0,C 180,E1 -14706.359,E2 -14706.359} C_VEL
LIN {X 0,Y 326.551,Z 162.805,A -85,B 0,C 180,E1 -14710.214,E2 -14710.214} C_VEL
LIN {X 0,Y 326.554,Z 162.807,A -85,B 0,C 180,E1 -14713.526,E2 -14713.526} C_VEL
LIN {X 0,Y 326.567,Z 162.809,A -85,B 0,C 180,E1 -14717.029,E2 -14717.029} C_VEL
LIN {X 0,Y 326.576,Z 162.804,A -85,B 0,C 180,E1 -14721.386,E2 -14721.386} C_VEL
LIN {X 0,Y 326.613,Z 162.803,A -85,B 0,C 180,E1 -14724.852,E2 -14724.852} C_VEL
LIN {X 0,Y 326.603,Z 162.799,A -85,B 0,C 180,E1 -14727.456,E2 -14727.456} C_VEL
LIN {X 0,Y 326.61,Z 162.8,A -85,B 0,C 180,E1 -14730.337,E2 -14730.337} C_VEL
LIN {X 0,Y 326.595,Z 162.804,A -85,B 0,C 180,E1 -14734.509,E2 -14734.509} C_VEL
LIN {X 0,Y 326.603,Z 162.804,A -85,B 0,C 180,E1 -14738.543,E2 -14738.543} C_VEL
LIN {X 0,Y 326.627,Z 162.801,A -85,B 0,C 180,E1 -14742.469,E2 -14742.469} C_VEL
LIN {X 0,Y 326.737,Z 162.787,A -85,B 0,C 180,E1 -14746.314,E2 -14746.314} C_VEL
LIN {X 0,Y 326.776,Z 162.781,A -85,B 0,C 180,E1 -14750.093,E2 -14750.093} C_VEL
LIN {X 0,Y 326.935,Z 162.76,A -85,B 0,C 180,E1 -14753.83,E2 -14753.83} C_VEL
LIN {X 0,Y 326.997,Z 162.751,A -85,B 0,C 180,E1 -14757.537,E2 -14757.537} C_VEL
LIN {X 0,Y 327.023,Z 162.747,A -85,B 0,C 180,E1 -14761.232,E2 -14761.232} C_VEL
LIN {X 0,Y 326.732,Z 162.786,A -85,B 0,C 180,E1 -14763.7,E2 -14763.7} C_VEL
LIN {X 0,Y 326.935,Z 162.761,A -85,B 0,C 180,E1 -14766.171,E2 -14766.171} C_VEL
LIN {X 0,Y 326.777,Z 162.782,A -85,B 0,C 180,E1 -14769.908,E2 -14769.908} C_VEL
LIN {X 0,Y 326.739,Z 162.787,A -85,B 0,C 180,E1 -14773.687,E2 -14773.687} C_VEL
LIN {X 0,Y 326.624,Z 162.8,A -85,B 0,C 180,E1 -14777.533,E2 -14777.533} C_VEL
LIN {X 0,Y 326.599,Z 162.804,A -85,B 0,C 180,E1 -14781.459,E2 -14781.459} C_VEL
LIN {X 0,Y 326.597,Z 162.805,A -85,B 0,C 180,E1 -14785.492,E2 -14785.492} C_VEL
LIN {X 0,Y 326.587,Z 162.801,A -85,B 0,C 180,E1 -14788.258,E2 -14788.258} C_VEL
LIN {X 0,Y 326.571,Z 162.806,A -85,B 0,C 180,E1 -14791.098,E2 -14791.098} C_VEL
LIN {X 0,Y 326.605,Z 162.799,A -85,B 0,C 180,E1 -14794.02,E2 -14794.02} C_VEL
LIN {X 0,Y 326.62,Z 162.802,A -85,B 0,C 180,E1 -14797.238,E2 -14797.238} C_VEL
LIN {X 0,Y 326.542,Z 162.812,A -85,B 0,C 180,E1 -14801.125,E2 -14801.125} C_VEL
LIN {X 0,Y 326.558,Z 162.806,A -85,B 0,C 180,E1 -14803.527,E2 -14803.527} C_VEL
LIN {X 0,Y 326.571,Z 162.808,A -85,B 0,C 180,E1 -14807.03,E2 -14807.03} C_VEL
LIN {X 0,Y 326.581,Z 162.803,A -85,B 0,C 180,E1 -14811.386,E2 -14811.386} C_VEL
LIN {X 0,Y 326.619,Z 162.803,A -85,B 0,C 180,E1 -14814.852,E2 -14814.852} C_VEL
LIN {X 0,Y 326.605,Z 162.803,A -85,B 0,C 180,E1 -14817.456,E2 -14817.456} C_VEL
LIN {X 0,Y 326.656,Z 162.874,A -85,B 0,C 180,E1 -14819.287,E2 -14819.287} C_VEL
LIN {X 0,Y 329.315,Z 175.946,A -85,B 0,C 180,E1 -14823.032,E2 -14823.032} C_VEL
LIN {X 0,Y 330.412,Z 182.451,A -85,B 0,C 180,E1 -14824.824,E2 -14824.824} C_VEL
LIN {X 0,Y 329.755,Z 189.127,A -85,B 0,C 180,E1 -14826.525,E2 -14826.525} C_VEL
LIN {X 0,Y 335.214,Z 226.877,A -85,B 0,C 180,E1 -14827.802,E2 -14827.802} C_VEL
LIN {X 0,Y 333.471,Z 297.568,A -85,B 0,C 180,E1 -14829.49,E2 -14829.49} C_VEL
LIN {X 0,Y 332.81,Z 311.078,A -85,B 0,C 180,E1 -14830.052,E2 -14830.052} C_VEL
LIN {X 0,Y 331.801,Z 323.967,A -85,B 0,C 180,E1 -14830.834,E2 -14830.834} C_VEL
LIN {X 0,Y 330.661,Z 336.573,A -85,B 0,C 180,E1 -14831.89,E2 -14831.89} C_VEL
LIN {X 0,Y 329.425,Z 347.85,A -85,B 0,C 180,E1 -14833.102,E2 -14833.102} C_VEL
LIN {X 0,Y 328.454,Z 358.093,A -85,B 0,C 180,E1 -14834.495,E2 -14834.495} C_VEL
LIN {X 0,Y 327.447,Z 367.236,A -85,B 0,C 180,E1 -14836.027,E2 -14836.027} C_VEL
LIN {X 0,Y 326.443,Z 376.2,A -85,B 0,C 180,E1 -14837.883,E2 -14837.883} C_VEL
LIN {X 0,Y 325.744,Z 383.347,A -85,B 0,C 180,E1 -14839.747,E2 -14839.747} C_VEL
LIN {X 0,Y 325.237,Z 389.864,A -85,B 0,C 180,E1 -14841.926,E2 -14841.926} C_VEL
LIN {X 0,Y 325.007,Z 394.754,A -85,B 0,C 180,E1 -14844.108,E2 -14844.108} C_VEL
LIN {X 0,Y 324.9,Z 398.103,A -85,B 0,C 180,E1 -14846.279,E2 -14846.279} C_VEL
LIN {X 0,Y 324.838,Z 399.414,A -85,B 0,C 180,E1 -14847.52,E2 -14847.52} C_VEL
LIN {X 0,Y 324.834,Z 400.32,A -85,B 0,C 180,E1 -14848.76,E2 -14848.76} C_VEL
LIN {X 0,Y 324.876,Z 400.796,A -85,B 0,C 180,E1 -14850,E2 -14850} C_VEL
LIN {X 0,Y 324.822,Z 400.834,A -85,B 0,C 180,E1 -14851.24,E2 -14851.24} C_VEL
LIN {X 0,Y 324.834,Z 400.477,A -85,B 0,C 180,E1 -14852.48,E2 -14852.48} C_VEL
LIN {X 0,Y 324.874,Z 399.725,A -85,B 0,C 180,E1 -14853.721,E2 -14853.721} C_VEL
LIN {X 0,Y 324.91,Z 397.614,A -85,B 0,C 180,E1 -14855.723,E2 -14855.723} C_VEL
LIN {X 0,Y 325.182,Z 394.869,A -85,B 0,C 180,E1 -14857.45,E2 -14857.45} C_VEL
LIN {X 0,Y 325.602,Z 390.916,A -85,B 0,C 180,E1 -14859.316,E2 -14859.316} C_VEL
LIN {X 0,Y 326.336,Z 385.825,A -85,B 0,C 180,E1 -14861.176,E2 -14861.176} C_VEL
LIN {X 0,Y 327.244,Z 379.45,A -85,B 0,C 180,E1 -14863.032,E2 -14863.032} C_VEL
LIN {X 0,Y 328.681,Z 371.509,A -85,B 0,C 180,E1 -14864.867,E2 -14864.867} C_VEL
LIN {X 0,Y 329.843,Z 362.889,A -85,B 0,C 180,E1 -14866.499,E2 -14866.499} C_VEL
LIN {X 0,Y 331.443,Z 352.585,A -85,B 0,C 180,E1 -14868.066,E2 -14868.066} C_VEL
LIN {X 0,Y 333.165,Z 341.389,A -85,B 0,C 180,E1 -14869.404,E2 -14869.404} C_VEL
LIN {X 0,Y 334.743,Z 328.773,A -85,B 0,C 180,E1 -14870.589,E2 -14870.589} C_VEL
LIN {X 0,Y 336.081,Z 316.253,A -85,B 0,C 180,E1 -14871.466,E2 -14871.466} C_VEL
LIN {X 0,Y 337.191,Z 303.186,A -85,B 0,C 180,E1 -14872.115,E2 -14872.115} C_VEL
LIN {X 0,Y 337.897,Z 289.465,A -85,B 0,C 180,E1 -14872.549,E2 -14872.549} C_VEL
LIN {X 0,Y 339.689,Z 226.404,A -85,B 0,C 180,E1 -14874.087,E2 -14874.087} C_VEL
LIN {X 0,Y 336.218,Z 205.211,A -85,B 0,C 180,E1 -14875.012,E2 -14875.012} C_VEL
LIN {X 0,Y 332.626,Z 189.554,A -85,B 0,C 180,E1 -14875.82,E2 -14875.82} C_VEL
LIN {X 0,Y 332.063,Z 187.286,A -85,B 0,C 180,E1 -14875.976,E2 -14875.976} C_VEL
LIN {X 0,Y 329.885,Z 176.07,A -85,B 0,C 180,E1 -14879.34,E2 -14879.34} C_VEL
LIN {X 0,Y 327.858,Z 167.661,A -85,B 0,C 180,E1 -14882.043,E2 -14882.043} C_VEL
LIN {X 0,Y 326.589,Z 162.805,A -85,B 0,C 180,E1 -14883.723,E2 -14883.723} C_VEL
LIN {X 0,Y 326.621,Z 162.802,A -85,B 0,C 180,E1 -14887.236,E2 -14887.236} C_VEL
LIN {X 0,Y 326.542,Z 162.814,A -85,B 0,C 180,E1 -14891.123,E2 -14891.123} C_VEL
LIN {X 0,Y 326.556,Z 162.813,A -85,B 0,C 180,E1 -14893.525,E2 -14893.525} C_VEL
LIN {X 0,Y 326.569,Z 162.804,A -85,B 0,C 180,E1 -14897.028,E2 -14897.028} C_VEL
LIN {X 0,Y 326.568,Z 162.802,A -85,B 0,C 180,E1 -14900.781,E2 -14900.781} C_VEL
LIN {X 0,Y 326.607,Z 162.799,A -85,B 0,C 180,E1 -14904.479,E2 -14904.479} C_VEL
LIN {X 0,Y 326.604,Z 162.798,A -85,B 0,C 180,E1 -14907.455,E2 -14907.455} C_VEL
LIN {X 0,Y 326.584,Z 162.796,A -85,B 0,C 180,E1 -14910.333,E2 -14910.333} C_VEL
LIN {X 0,Y 326.591,Z 162.795,A -85,B 0,C 180,E1 -14913.133,E2 -14913.133} C_VEL
LIN {X 0,Y 326.586,Z 162.794,A -85,B 0,C 180,E1 -14917.21,E2 -14917.21} C_VEL
LIN {X 0,Y 326.623,Z 162.79,A -85,B 0,C 180,E1 -14921.216,E2 -14921.216} C_VEL
LIN {X 0,Y 326.72,Z 162.781,A -85,B 0,C 180,E1 -14925.459,E2 -14925.459} C_VEL
LIN {X 0,Y 326.748,Z 162.778,A -85,B 0,C 180,E1 -14928.838,E2 -14928.838} C_VEL
LIN {X 0,Y 326.906,Z 162.762,A -85,B 0,C 180,E1 -14932.588,E2 -14932.588} C_VEL
LIN {X 0,Y 326.736,Z 162.778,A -85,B 0,C 180,E1 -14935.064,E2 -14935.064} C_VEL
LIN {X 0,Y 327.001,Z 162.751,A -85,B 0,C 180,E1 -14937.536,E2 -14937.536} C_VEL
LIN {X 0,Y 327.021,Z 162.746,A -85,B 0,C 180,E1 -14941.231,E2 -14941.231} C_VEL
LIN {X 0,Y 326.74,Z 162.783,A -85,B 0,C 180,E1 -14943.699,E2 -14943.699} C_VEL
LIN {X 0,Y 326.913,Z 162.761,A -85,B 0,C 180,E1 -14946.45,E2 -14946.45} C_VEL
LIN {X 0,Y 326.774,Z 162.784,A -85,B 0,C 180,E1 -14949.907,E2 -14949.907} C_VEL
LIN {X 0,Y 326.729,Z 162.794,A -85,B 0,C 180,E1 -14954.172,E2 -14954.172} C_VEL
LIN {X 0,Y 326.742,Z 162.873,A -85,B 0,C 180,E1 -14954.334,E2 -14954.334} C_VEL
LIN {X 0,Y 329.213,Z 173.026,A -85,B 0,C 180,E1 -14957.79,E2 -14957.79} C_VEL
LIN {X 0,Y 336.949,Z 190.037,A -85,B 0,C 180,E1 -14959.103,E2 -14959.103} C_VEL
LIN {X 0,Y 338.847,Z 195.462,A -85,B 0,C 180,E1 -14959.443,E2 -14959.443} C_VEL
LIN {X 0,Y 340.448,Z 203.555,A -85,B 0,C 180,E1 -14959.823,E2 -14959.823} C_VEL
LIN {X 0,Y 337.859,Z 281.258,A -85,B 0,C 180,E1 -14961.737,E2 -14961.737} C_VEL
LIN {X 0,Y 337.02,Z 294.593,A -85,B 0,C 180,E1 -14962.302,E2 -14962.302} C_VEL
LIN {X 0,Y 336.06,Z 306.697,A -85,B 0,C 180,E1 -14963.052,E2 -14963.052} C_VEL
LIN {X 0,Y 334.826,Z 318.152,A -85,B 0,C 180,E1 -14963.996,E2 -14963.996} C_VEL
LIN {X 0,Y 333.274,Z 330.207,A -85,B 0,C 180,E1 -14965.278,E2 -14965.278} C_VEL
LIN {X 0,Y 331.653,Z 340.844,A -85,B 0,C 180,E1 -14966.712,E2 -14966.712} C_VEL
LIN {X 0,Y 330.104,Z 350.98,A -85,B 0,C 180,E1 -14968.448,E2 -14968.448} C_VEL
LIN {X 0,Y 328.749,Z 359.025,A -85,B 0,C 180,E1 -14970.157,E2 -14970.157} C_VEL
LIN {X 0,Y 327.504,Z 366.231,A -85,B 0,C 180,E1 -14972.083,E2 -14972.083} C_VEL
LIN {X 0,Y 326.54,Z 371.963,A -85,B 0,C 180,E1 -14974.027,E2 -14974.027} C_VEL
LIN {X 0,Y 325.732,Z 377.033,A -85,B 0,C 180,E1 -14976.294,E2 -14976.294} C_VEL
LIN {X 0,Y 325.283,Z 379.774,A -85,B 0,C 180,E1 -14978.007,E2 -14978.007} C_VEL
LIN {X 0,Y 324.881,Z 382.286,A -85,B 0,C 180,E1 -14980.464,E2 -14980.464} C_VEL
LIN {X 0,Y 324.626,Z 383.152,A -85,B 0,C 180,E1 -14982.602,E2 -14982.602} C_VEL
LIN {X 0,Y 324.619,Z 382.955,A -85,B 0,C 180,E1 -14984.403,E2 -14984.403} C_VEL
LIN {X 0,Y 324.681,Z 381.943,A -85,B 0,C 180,E1 -14986.16,E2 -14986.16} C_VEL
LIN {X 0,Y 324.836,Z 380.113,A -85,B 0,C 180,E1 -14987.88,E2 -14987.88} C_VEL
LIN {X 0,Y 325.048,Z 377.519,A -85,B 0,C 180,E1 -14989.562,E2 -14989.562} C_VEL
LIN {X 0,Y 325.401,Z 374.133,A -85,B 0,C 180,E1 -14991.22,E2 -14991.22} C_VEL
LIN {X 0,Y 325.96,Z 368.533,A -85,B 0,C 180,E1 -14993.318,E2 -14993.318} C_VEL
LIN {X 0,Y 326.555,Z 362.192,A -85,B 0,C 180,E1 -14995.175,E2 -14995.175} C_VEL
LIN {X 0,Y 327.368,Z 355.087,A -85,B 0,C 180,E1 -14996.851,E2 -14996.851} C_VEL
LIN {X 0,Y 328.429,Z 345.969,A -85,B 0,C 180,E1 -14998.585,E2 -14998.585} C_VEL
LIN {X 0,Y 329.467,Z 336.198,A -85,B 0,C 180,E1 -15000.092,E2 -15000.092} C_VEL
LIN {X 0,Y 330.558,Z 325.492,A -85,B 0,C 180,E1 -15001.422,E2 -15001.422} C_VEL
LIN {X 0,Y 331.647,Z 312.965,A -85,B 0,C 180,E1 -15002.636,E2 -15002.636} C_VEL
LIN {X 0,Y 332.616,Z 301.074,A -85,B 0,C 180,E1 -15003.515,E2 -15003.515} C_VEL
LIN {X 0,Y 333.208,Z 288.842,A -85,B 0,C 180,E1 -15004.182,E2 -15004.182} C_VEL
LIN {X 0,Y 333.775,Z 275.1,A -85,B 0,C 180,E1 -15004.662,E2 -15004.662} C_VEL
LIN {X 0,Y 335.487,Z 200.627,A -85,B 0,C 180,E1 -15006.424,E2 -15006.424} C_VEL
LIN {X 0,Y 332.023,Z 182.622,A -85,B 0,C 180,E1 -15007.084,E2 -15007.084} C_VEL
LIN {X 0,Y 328.451,Z 171.929,A -85,B 0,C 180,E1 -15007.596,E2 -15007.596} C_VEL
LIN {X 0,Y 326.631,Z 162.801,A -85,B 0,C 180,E1 -15010.437,E2 -15010.437} C_VEL
LIN {X 0,Y 326.671,Z 162.791,A -85,B 0,C 180,E1 -15013.759,E2 -15013.759} C_VEL
LIN {X 0,Y 326.738,Z 162.787,A -85,B 0,C 180,E1 -15016.314,E2 -15016.314} C_VEL
LIN {X 0,Y 326.778,Z 162.781,A -85,B 0,C 180,E1 -15020.093,E2 -15020.093} C_VEL
LIN {X 0,Y 326.938,Z 162.759,A -85,B 0,C 180,E1 -15023.83,E2 -15023.83} C_VEL
LIN {X 0,Y 327.005,Z 162.75,A -85,B 0,C 180,E1 -15027.537,E2 -15027.537} C_VEL
LIN {X 0,Y 327.024,Z 162.747,A -85,B 0,C 180,E1 -15031.232,E2 -15031.232} C_VEL
LIN {X 0,Y 326.734,Z 162.785,A -85,B 0,C 180,E1 -15033.7,E2 -15033.7} C_VEL
LIN {X 0,Y 326.936,Z 162.761,A -85,B 0,C 180,E1 -15036.17,E2 -15036.17} C_VEL
LIN {X 0,Y 326.778,Z 162.783,A -85,B 0,C 180,E1 -15039.907,E2 -15039.907} C_VEL
LIN {X 0,Y 326.739,Z 162.787,A -85,B 0,C 180,E1 -15043.686,E2 -15043.686} C_VEL
LIN {X 0,Y 326.624,Z 162.8,A -85,B 0,C 180,E1 -15047.532,E2 -15047.532} C_VEL
LIN {X 0,Y 326.603,Z 162.803,A -85,B 0,C 180,E1 -15051.458,E2 -15051.458} C_VEL
LIN {X 0,Y 326.595,Z 162.805,A -85,B 0,C 180,E1 -15055.491,E2 -15055.491} C_VEL
LIN {X 0,Y 326.585,Z 162.801,A -85,B 0,C 180,E1 -15058.257,E2 -15058.257} C_VEL
LIN {X 0,Y 326.568,Z 162.806,A -85,B 0,C 180,E1 -15061.097,E2 -15061.097} C_VEL
LIN {X 0,Y 326.603,Z 162.799,A -85,B 0,C 180,E1 -15064.02,E2 -15064.02} C_VEL
LIN {X 0,Y 326.587,Z 162.801,A -85,B 0,C 180,E1 -15066.359,E2 -15066.359} C_VEL
LIN {X 0,Y 325.934,Z 162.887,A -85,B 0,C 180,E1 -15067.388,E2 -15067.388} C_VEL
LIN {X 0,Y 323.069,Z 163.244,A -85,B 0,C 180,E1 -15069.062,E2 -15069.062} C_VEL
LIN {X 0,Y 320.629,Z 163.547,A -85,B 0,C 180,E1 -15070.419,E2 -15070.419} C_VEL
LIN {X 0,Y 319.579,Z 163.676,A -85,B 0,C 180,E1 -15071.469,E2 -15071.469} C_VEL
LIN {X 0,Y 319.493,Z 163.684,A -85,B 0,C 180,E1 -15071.825,E2 -15071.825} C_VEL
LIN {X 0,Y 319.481,Z 163.689,A -85,B 0,C 180,E1 -15075.257,E2 -15075.257} C_VEL
LIN {X 0,Y 319.499,Z 163.685,A -85,B 0,C 180,E1 -15078.408,E2 -15078.408} C_VEL
LIN {X 0,Y 319.526,Z 163.68,A -85,B 0,C 180,E1 -15081.986,E2 -15081.986} C_VEL
LIN {X 0,Y 319.554,Z 163.679,A -85,B 0,C 180,E1 -15085.123,E2 -15085.123} C_VEL
LIN {X 0,Y 319.519,Z 163.681,A -85,B 0,C 180,E1 -15088.137,E2 -15088.137} C_VEL
LIN {X 0,Y 319.564,Z 163.676,A -85,B 0,C 180,E1 -15091.605,E2 -15091.605} C_VEL
LIN {X 0,Y 319.521,Z 163.682,A -85,B 0,C 180,E1 -15095.298,E2 -15095.298} C_VEL
LIN {X 0,Y 319.558,Z 163.677,A -85,B 0,C 180,E1 -15098.046,E2 -15098.046} C_VEL
LIN {X 0,Y 319.582,Z 163.674,A -85,B 0,C 180,E1 -15102.069,E2 -15102.069} C_VEL
LIN {X 0,Y 319.704,Z 163.66,A -85,B 0,C 180,E1 -15106.007,E2 -15106.007} C_VEL
LIN {X 0,Y 319.729,Z 163.657,A -85,B 0,C 180,E1 -15109.872,E2 -15109.872} C_VEL
LIN {X 0,Y 319.892,Z 163.635,A -85,B 0,C 180,E1 -15113.694,E2 -15113.694} C_VEL
LIN {X 0,Y 319.943,Z 163.629,A -85,B 0,C 180,E1 -15117.483,E2 -15117.483} C_VEL
LIN {X 0,Y 319.992,Z 163.623,A -85,B 0,C 180,E1 -15121.259,E2 -15121.259} C_VEL
LIN {X 0,Y 319.709,Z 163.657,A -85,B 0,C 180,E1 -15125.045,E2 -15125.045} C_VEL
LIN {X 0,Y 319.848,Z 163.642,A -85,B 0,C 180,E1 -15127.576,E2 -15127.576} C_VEL
LIN {X 0,Y 319.707,Z 163.66,A -85,B 0,C 180,E1 -15131.411,E2 -15131.411} C_VEL
LIN {X 0,Y 319.66,Z 163.664,A -85,B 0,C 180,E1 -15134.677,E2 -15134.677} C_VEL
LIN {X 0,Y 319.597,Z 163.672,A -85,B 0,C 180,E1 -15138.992,E2 -15138.992} C_VEL
LIN {X 0,Y 319.578,Z 163.674,A -85,B 0,C 180,E1 -15142.537,E2 -15142.537} C_VEL
LIN {X 0,Y 319.546,Z 163.679,A -85,B 0,C 180,E1 -15146.096,E2 -15146.096} C_VEL
LIN {X 0,Y 319.522,Z 163.683,A -85,B 0,C 180,E1 -15148.941,E2 -15148.941} C_VEL
LIN {X 0,Y 319.522,Z 163.682,A -85,B 0,C 180,E1 -15151.863,E2 -15151.863} C_VEL
LIN {X 0,Y 319.577,Z 163.677,A -85,B 0,C 180,E1 -15155.543,E2 -15155.543} C_VEL
LIN {X 0,Y 319.527,Z 163.682,A -85,B 0,C 180,E1 -15159.663,E2 -15159.663} C_VEL
LIN {X 0,Y 319.517,Z 163.684,A -85,B 0,C 180,E1 -15163.46,E2 -15163.46} C_VEL
LIN {X 0,Y 319.55,Z 163.683,A -85,B 0,C 180,E1 -15167.016,E2 -15167.016} C_VEL
LIN {X 0,Y 319.545,Z 163.679,A -85,B 0,C 180,E1 -15170.371,E2 -15170.371} C_VEL
LIN {X 0,Y 319.579,Z 163.676,A -85,B 0,C 180,E1 -15174.458,E2 -15174.458} C_VEL
LIN {X 0,Y 319.534,Z 163.682,A -85,B 0,C 180,E1 -15178.139,E2 -15178.139} C_VEL
LIN {X 0,Y 319.583,Z 163.822,A -85,B 0,C 180,E1 -15178.981,E2 -15178.981} C_VEL
LIN {X 0,Y 322.233,Z 176.637,A -85,B 0,C 180,E1 -15182.741,E2 -15182.741} C_VEL
LIN {X 0,Y 323.447,Z 184.445,A -85,B 0,C 180,E1 -15184.931,E2 -15184.931} C_VEL
LIN {X 0,Y 322.89,Z 188.898,A -85,B 0,C 180,E1 -15186.089,E2 -15186.089} C_VEL
LIN {X 0,Y 328.441,Z 227.105,A -85,B 0,C 180,E1 -15187.428,E2 -15187.428} C_VEL
LIN {X 0,Y 326.65,Z 297.942,A -85,B 0,C 180,E1 -15189.165,E2 -15189.165} C_VEL
LIN {X 0,Y 325.895,Z 311.997,A -85,B 0,C 180,E1 -15189.775,E2 -15189.775} C_VEL
LIN {X 0,Y 324.879,Z 324.518,A -85,B 0,C 180,E1 -15190.573,E2 -15190.573} C_VEL
LIN {X 0,Y 323.713,Z 336.973,A -85,B 0,C 180,E1 -15191.651,E2 -15191.651} C_VEL
LIN {X 0,Y 322.448,Z 348.138,A -85,B 0,C 180,E1 -15192.888,E2 -15192.888} C_VEL
LIN {X 0,Y 321.424,Z 358.365,A -85,B 0,C 180,E1 -15194.325,E2 -15194.325} C_VEL
LIN {X 0,Y 320.319,Z 368.187,A -85,B 0,C 180,E1 -15196.034,E2 -15196.034} C_VEL
LIN {X 0,Y 319.482,Z 375.585,A -85,B 0,C 180,E1 -15197.615,E2 -15197.615} C_VEL
LIN {X 0,Y 318.723,Z 382.84,A -85,B 0,C 180,E1 -15199.519,E2 -15199.519} C_VEL
LIN {X 0,Y 318.186,Z 389.423,A -85,B 0,C 180,E1 -15201.745,E2 -15201.745} C_VEL
LIN {X 0,Y 317.924,Z 393.741,A -85,B 0,C 180,E1 -15203.654,E2 -15203.654} C_VEL
LIN {X 0,Y 317.816,Z 396.018,A -85,B 0,C 180,E1 -15204.925,E2 -15204.925} C_VEL
LIN {X 0,Y 317.807,Z 397.799,A -85,B 0,C 180,E1 -15206.196,E2 -15206.196} C_VEL
LIN {X 0,Y 317.76,Z 399.136,A -85,B 0,C 180,E1 -15207.465,E2 -15207.465} C_VEL
LIN {X 0,Y 317.746,Z 400.065,A -85,B 0,C 180,E1 -15208.732,E2 -15208.732} C_VEL
LIN {X 0,Y 317.783,Z 400.583,A -85,B 0,C 180,E1 -15210,E2 -15210} C_VEL
LIN {X 0,Y 317.734,Z 400.647,A -85,B 0,C 180,E1 -15211.267,E2 -15211.267} C_VEL
LIN {X 0,Y 317.755,Z 400.312,A -85,B 0,C 180,E1 -15212.535,E2 -15212.535} C_VEL
LIN {X 0,Y 317.784,Z 399.58,A -85,B 0,C 180,E1 -15213.804,E2 -15213.804} C_VEL
LIN {X 0,Y 317.826,Z 397.71,A -85,B 0,C 180,E1 -15215.685,E2 -15215.685} C_VEL
LIN {X 0,Y 318.108,Z 394.81,A -85,B 0,C 180,E1 -15217.617,E2 -15217.617} C_VEL
LIN {X 0,Y 318.586,Z 390.912,A -85,B 0,C 180,E1 -15219.523,E2 -15219.523} C_VEL
LIN {X 0,Y 319.353,Z 385.888,A -85,B 0,C 180,E1 -15221.423,E2 -15221.423} C_VEL
LIN {X 0,Y 320.332,Z 379.589,A -85,B 0,C 180,E1 -15223.318,E2 -15223.318} C_VEL
LIN {X 0,Y 321.828,Z 371.753,A -85,B 0,C 180,E1 -15225.191,E2 -15225.191} C_VEL
LIN {X 0,Y 322.998,Z 363.613,A -85,B 0,C 180,E1 -15226.786,E2 -15226.786} C_VEL
LIN {X 0,Y 324.732,Z 353.008,A -85,B 0,C 180,E1 -15228.452,E2 -15228.452} C_VEL
LIN {X 0,Y 326.528,Z 342.009,A -85,B 0,C 180,E1 -15229.815,E2 -15229.815} C_VEL
LIN {X 0,Y 328.156,Z 329.586,A -85,B 0,C 180,E1 -15231.022,E2 -15231.022} C_VEL
LIN {X 0,Y 329.551,Z 317.551,A -85,B 0,C 180,E1 -15231.913,E2 -15231.913} C_VEL
LIN {X 0,Y 330.751,Z 304.321,A -85,B 0,C 180,E1 -15232.61,E2 -15232.61} C_VEL
LIN {X 0,Y 331.546,Z 291.577,A -85,B 0,C 180,E1 -15233.047,E2 -15233.047} C_VEL
LIN {X 0,Y 333.482,Z 227.465,A -85,B 0,C 180,E1 -15234.653,E2 -15234.653} C_VEL
LIN {X 0,Y 330.315,Z 207.828,A -85,B 0,C 180,E1 -15235.533,E2 -15235.533} C_VEL
LIN {X 0,Y 326.862,Z 192.248,A -85,B 0,C 180,E1 -15236.363,E2 -15236.363} C_VEL
LIN {X 0,Y 324.912,Z 187.039,A -85,B 0,C 180,E1 -15236.764,E2 -15236.764} C_VEL
LIN {X 0,Y 322.827,Z 176.484,A -85,B 0,C 180,E1 -15240.046,E2 -15240.046} C_VEL
LIN {X 0,Y 320.393,Z 167.009,A -85,B 0,C 180,E1 -15243.256,E2 -15243.256} C_VEL
LIN {X 0,Y 319.57,Z 163.68,A -85,B 0,C 180,E1 -15244.491,E2 -15244.491} C_VEL
LIN {X 0,Y 319.522,Z 163.687,A -85,B 0,C 180,E1 -15248.014,E2 -15248.014} C_VEL
LIN {X 0,Y 319.502,Z 163.692,A -85,B 0,C 180,E1 -15251.591,E2 -15251.591} C_VEL
LIN {X 0,Y 319.483,Z 163.689,A -85,B 0,C 180,E1 -15254.743,E2 -15254.743} C_VEL
LIN {X 0,Y 319.547,Z 163.679,A -85,B 0,C 180,E1 -15257.015,E2 -15257.015} C_VEL
LIN {X 0,Y 319.512,Z 163.68,A -85,B 0,C 180,E1 -15260.365,E2 -15260.365} C_VEL
LIN {X 0,Y 319.575,Z 163.674,A -85,B 0,C 180,E1 -15264.457,E2 -15264.457} C_VEL
LIN {X 0,Y 319.52,Z 163.682,A -85,B 0,C 180,E1 -15268.136,E2 -15268.136} C_VEL
LIN {X 0,Y 319.563,Z 163.677,A -85,B 0,C 180,E1 -15271.604,E2 -15271.604} C_VEL
LIN {X 0,Y 319.535,Z 163.682,A -85,B 0,C 180,E1 -15275.298,E2 -15275.298} C_VEL
LIN {X 0,Y 319.557,Z 163.672,A -85,B 0,C 180,E1 -15278.044,E2 -15278.044} C_VEL
LIN {X 0,Y 319.57,Z 163.672,A -85,B 0,C 180,E1 -15282.067,E2 -15282.067} C_VEL
LIN {X 0,Y 319.704,Z 163.658,A -85,B 0,C 180,E1 -15286.006,E2 -15286.006} C_VEL
LIN {X 0,Y 319.728,Z 163.658,A -85,B 0,C 180,E1 -15289.871,E2 -15289.871} C_VEL
LIN {X 0,Y 319.89,Z 163.64,A -85,B 0,C 180,E1 -15293.693,E2 -15293.693} C_VEL
LIN {X 0,Y 319.947,Z 163.629,A -85,B 0,C 180,E1 -15297.482,E2 -15297.482} C_VEL
LIN {X 0,Y 319.991,Z 163.622,A -85,B 0,C 180,E1 -15301.258,E2 -15301.258} C_VEL
LIN {X 0,Y 319.69,Z 163.661,A -85,B 0,C 180,E1 -15303.781,E2 -15303.781} C_VEL
LIN {X 0,Y 319.878,Z 163.639,A -85,B 0,C 180,E1 -15306.431,E2 -15306.431} C_VEL
LIN {X 0,Y 319.727,Z 163.663,A -85,B 0,C 180,E1 -15310.128,E2 -15310.128} C_VEL
LIN {X 0,Y 319.709,Z 163.721,A -85,B 0,C 180,E1 -15313.587,E2 -15313.587} C_VEL
LIN {X 0,Y 322.094,Z 173.34,A -85,B 0,C 180,E1 -15316.992,E2 -15316.992} C_VEL
LIN {X 0,Y 330.16,Z 190.537,A -85,B 0,C 180,E1 -15318.419,E2 -15318.419} C_VEL
LIN {X 0,Y 332.919,Z 197.81,A -85,B 0,C 180,E1 -15318.916,E2 -15318.916} C_VEL
LIN {X 0,Y 334.279,Z 205.128,A -85,B 0,C 180,E1 -15319.261,E2 -15319.261} C_VEL
LIN {X 0,Y 331.557,Z 281.683,A -85,B 0,C 180,E1 -15321.187,E2 -15321.187} C_VEL
LIN {X 0,Y 330.678,Z 295.025,A -85,B 0,C 180,E1 -15321.769,E2 -15321.769} C_VEL
LIN {X 0,Y 329.608,Z 307.518,A -85,B 0,C 180,E1 -15322.569,E2 -15322.569} C_VEL
LIN {X 0,Y 328.141,Z 319.942,A -85,B 0,C 180,E1 -15323.638,E2 -15323.638} C_VEL
LIN {X 0,Y 326.567,Z 331.627,A -85,B 0,C 180,E1 -15324.941,E2 -15324.941} C_VEL
LIN {X 0,Y 324.947,Z 341.479,A -85,B 0,C 180,E1 -15326.319,E2 -15326.319} C_VEL
LIN {X 0,Y 323.544,Z 350.356,A -85,B 0,C 180,E1 -15327.86,E2 -15327.86} C_VEL
LIN {X 0,Y 322.02,Z 358.853,A -85,B 0,C 180,E1 -15329.672,E2 -15329.672} C_VEL
LIN {X 0,Y 320.626,Z 366.485,A -85,B 0,C 180,E1 -15331.74,E2 -15331.74} C_VEL
LIN {X 0,Y 319.769,Z 371.297,A -85,B 0,C 180,E1 -15333.367,E2 -15333.367} C_VEL
LIN {X 0,Y 318.952,Z 375.981,A -85,B 0,C 180,E1 -15335.386,E2 -15335.386} C_VEL
LIN {X 0,Y 318.362,Z 379.401,A -85,B 0,C 180,E1 -15337.373,E2 -15337.373} C_VEL
LIN {X 0,Y 317.845,Z 382.195,A -85,B 0,C 180,E1 -15339.883,E2 -15339.883} C_VEL
LIN {X 0,Y 317.623,Z 383.143,A -85,B 0,C 180,E1 -15341.59,E2 -15341.59} C_VEL
LIN {X 0,Y 317.506,Z 383.372,A -85,B 0,C 180,E1 -15343.328,E2 -15343.328} C_VEL
LIN {X 0,Y 317.524,Z 382.829,A -85,B 0,C 180,E1 -15345.094,E2 -15345.094} C_VEL
LIN {X 0,Y 317.651,Z 381.423,A -85,B 0,C 180,E1 -15346.896,E2 -15346.896} C_VEL
LIN {X 0,Y 317.823,Z 379.091,A -85,B 0,C 180,E1 -15348.749,E2 -15348.749} C_VEL
LIN {X 0,Y 318.187,Z 375.746,A -85,B 0,C 180,E1 -15350.629,E2 -15350.629} C_VEL
LIN {X 0,Y 318.651,Z 371.191,A -85,B 0,C 180,E1 -15352.56,E2 -15352.56} C_VEL
LIN {X 0,Y 319.249,Z 365.202,A -85,B 0,C 180,E1 -15354.539,E2 -15354.539} C_VEL
LIN {X 0,Y 320.121,Z 357.476,A -85,B 0,C 180,E1 -15356.538,E2 -15356.538} C_VEL
LIN {X 0,Y 321.124,Z 348.901,A -85,B 0,C 180,E1 -15358.315,E2 -15358.315} C_VEL
LIN {X 0,Y 322.195,Z 339.549,A -85,B 0,C 180,E1 -15359.888,E2 -15359.888} C_VEL
LIN {X 0,Y 323.262,Z 329.654,A -85,B 0,C 180,E1 -15361.233,E2 -15361.233} C_VEL
LIN {X 0,Y 324.422,Z 317.31,A -85,B 0,C 180,E1 -15362.568,E2 -15362.568} C_VEL
LIN {X 0,Y 325.434,Z 305.484,A -85,B 0,C 180,E1 -15363.551,E2 -15363.551} C_VEL
LIN {X 0,Y 326.234,Z 292.055,A -85,B 0,C 180,E1 -15364.372,E2 -15364.372} C_VEL
LIN {X 0,Y 326.861,Z 278.786,A -85,B 0,C 180,E1 -15364.914,E2 -15364.914} C_VEL
LIN {X 0,Y 328.863,Z 202.187,A -85,B 0,C 180,E1 -15366.769,E2 -15366.769} C_VEL
LIN {X 0,Y 325.624,Z 185.048,A -85,B 0,C 180,E1 -15367.412,E2 -15367.412} C_VEL
LIN {X 0,Y 321.265,Z 172.146,A -85,B 0,C 180,E1 -15368.042,E2 -15368.042} C_VEL
LIN {X 0,Y 319.588,Z 163.678,A -85,B 0,C 180,E1 -15370.74,E2 -15370.74} C_VEL
LIN {X 0,Y 319.631,Z 163.671,A -85,B 0,C 180,E1 -15374.702,E2 -15374.702} C_VEL
LIN {X 0,Y 319.669,Z 163.663,A -85,B 0,C 180,E1 -15377.3,E2 -15377.3} C_VEL
LIN {X 0,Y 319.821,Z 163.644,A -85,B 0,C 180,E1 -15381.437,E2 -15381.437} C_VEL
LIN {X 0,Y 319.896,Z 163.636,A -85,B 0,C 180,E1 -15383.694,E2 -15383.694} C_VEL
LIN {X 0,Y 319.951,Z 163.628,A -85,B 0,C 180,E1 -15387.482,E2 -15387.482} C_VEL
LIN {X 0,Y 319.994,Z 163.623,A -85,B 0,C 180,E1 -15391.259,E2 -15391.259} C_VEL
LIN {X 0,Y 319.685,Z 163.664,A -85,B 0,C 180,E1 -15393.782,E2 -15393.782} C_VEL
LIN {X 0,Y 319.894,Z 163.637,A -85,B 0,C 180,E1 -15396.307,E2 -15396.307} C_VEL
LIN {X 0,Y 319.73,Z 163.658,A -85,B 0,C 180,E1 -15400.128,E2 -15400.128} C_VEL
LIN {X 0,Y 319.706,Z 163.662,A -85,B 0,C 180,E1 -15403.993,E2 -15403.993} C_VEL
LIN {X 0,Y 319.58,Z 163.677,A -85,B 0,C 180,E1 -15407.931,E2 -15407.931} C_VEL
LIN {X 0,Y 319.558,Z 163.679,A -85,B 0,C 180,E1 -15411.955,E2 -15411.955} C_VEL
LIN {X 0,Y 319.545,Z 163.679,A -85,B 0,C 180,E1 -15416.096,E2 -15416.096} C_VEL
LIN {X 0,Y 319.52,Z 163.683,A -85,B 0,C 180,E1 -15418.94,E2 -15418.94} C_VEL
LIN {X 0,Y 319.52,Z 163.682,A -85,B 0,C 180,E1 -15421.863,E2 -15421.863} C_VEL
LIN {X 0,Y 319.575,Z 163.677,A -85,B 0,C 180,E1 -15425.543,E2 -15425.543} C_VEL
LIN {X 0,Y 319.524,Z 163.682,A -85,B 0,C 180,E1 -15429.662,E2 -15429.662} C_VEL
LIN {X 0,Y 319.493,Z 163.684,A -85,B 0,C 180,E1 -15431.825,E2 -15431.825} C_VEL
LIN {X 0,Y 318.813,Z 163.772,A -85,B 0,C 180,E1 -15432.877,E2 -15432.877} C_VEL
LIN {X 0,Y 315.927,Z 164.129,A -85,B 0,C 180,E1 -15434.587,E2 -15434.587} C_VEL
LIN {X 0,Y 313.509,Z 164.429,A -85,B 0,C 180,E1 -15435.974,E2 -15435.974} C_VEL
LIN {X 0,Y 312.51,Z 164.56,A -85,B 0,C 180,E1 -15437.049,E2 -15437.049} C_VEL
LIN {X 0,Y 312.449,Z 164.562,A -85,B 0,C 180,E1 -15437.412,E2 -15437.412} C_VEL
LIN {X 0,Y 312.489,Z 164.562,A -85,B 0,C 180,E1 -15440.971,E2 -15440.971} C_VEL
LIN {X 0,Y 312.525,Z 164.552,A -85,B 0,C 180,E1 -15444.22,E2 -15444.22} C_VEL
LIN {X 0,Y 312.497,Z 164.555,A -85,B 0,C 180,E1 -15447.334,E2 -15447.334} C_VEL
LIN {X 0,Y 312.5,Z 164.556,A -85,B 0,C 180,E1 -15451.293,E2 -15451.293} C_VEL
LIN {X 0,Y 312.512,Z 164.559,A -85,B 0,C 180,E1 -15454.705,E2 -15454.705} C_VEL
LIN {X 0,Y 312.534,Z 164.551,A -85,B 0,C 180,E1 -15457.526,E2 -15457.526} C_VEL
LIN {X 0,Y 312.542,Z 164.548,A -85,B 0,C 180,E1 -15461.651,E2 -15461.651} C_VEL
LIN {X 0,Y 312.647,Z 164.537,A -85,B 0,C 180,E1 -15465.685,E2 -15465.685} C_VEL
LIN {X 0,Y 312.679,Z 164.534,A -85,B 0,C 180,E1 -15469.642,E2 -15469.642} C_VEL
LIN {X 0,Y 312.834,Z 164.513,A -85,B 0,C 180,E1 -15473.551,E2 -15473.551} C_VEL
LIN {X 0,Y 312.891,Z 164.506,A -85,B 0,C 180,E1 -15477.426,E2 -15477.426} C_VEL
LIN {X 0,Y 312.944,Z 164.505,A -85,B 0,C 180,E1 -15480.001,E2 -15480.001} C_VEL
LIN {X 0,Y 312.891,Z 164.508,A -85,B 0,C 180,E1 -15482.575,E2 -15482.575} C_VEL
LIN {X 0,Y 312.834,Z 164.514,A -85,B 0,C 180,E1 -15486.45,E2 -15486.45} C_VEL
LIN {X 0,Y 312.68,Z 164.534,A -85,B 0,C 180,E1 -15490.359,E2 -15490.359} C_VEL
LIN {X 0,Y 312.648,Z 164.538,A -85,B 0,C 180,E1 -15494.316,E2 -15494.316} C_VEL
LIN {X 0,Y 312.538,Z 164.551,A -85,B 0,C 180,E1 -15498.35,E2 -15498.35} C_VEL
LIN {X 0,Y 312.536,Z 164.551,A -85,B 0,C 180,E1 -15502.475,E2 -15502.475} C_VEL
LIN {X 0,Y 312.504,Z 164.557,A -85,B 0,C 180,E1 -15505.899,E2 -15505.899} C_VEL
LIN {X 0,Y 312.466,Z 164.563,A -85,B 0,C 180,E1 -15509.659,E2 -15509.659} C_VEL
LIN {X 0,Y 312.518,Z 164.554,A -85,B 0,C 180,E1 -15513.689,E2 -15513.689} C_VEL
LIN {X 0,Y 312.511,Z 164.558,A -85,B 0,C 180,E1 -15517.388,E2 -15517.388} C_VEL
LIN {X 0,Y 312.439,Z 164.565,A -85,B 0,C 180,E1 -15520.718,E2 -15520.718} C_VEL
LIN {X 0,Y 312.449,Z 164.562,A -85,B 0,C 180,E1 -15524.211,E2 -15524.211} C_VEL
LIN {X 0,Y 312.453,Z 164.562,A -85,B 0,C 180,E1 -15527.926,E2 -15527.926} C_VEL
LIN {X 0,Y 312.483,Z 164.558,A -85,B 0,C 180,E1 -15531.923,E2 -15531.923} C_VEL
LIN {X 0,Y 312.53,Z 164.553,A -85,B 0,C 180,E1 -15534.22,E2 -15534.22} C_VEL
LIN {X 0,Y 312.487,Z 164.56,A -85,B 0,C 180,E1 -15538.085,E2 -15538.085} C_VEL
LIN {X 0,Y 312.529,Z 164.722,A -85,B 0,C 180,E1 -15538.649,E2 -15538.649} C_VEL
LIN {X 0,Y 315.116,Z 177.077,A -85,B 0,C 180,E1 -15542.368,E2 -15542.368} C_VEL
LIN {X 0,Y 316.444,Z 185.142,A -85,B 0,C 180,E1 -15544.689,E2 -15544.689} C_VEL
LIN {X 0,Y 316.035,Z 188.724,A -85,B 0,C 180,E1 -15545.646,E2 -15545.646} C_VEL
LIN {X 0,Y 321.69,Z 228.255,A -85,B 0,C 180,E1 -15547.063,E2 -15547.063} C_VEL
LIN {X 0,Y 319.891,Z 297.233,A -85,B 0,C 180,E1 -15548.788,E2 -15548.788} C_VEL
LIN {X 0,Y 319.169,Z 310.698,A -85,B 0,C 180,E1 -15549.371,E2 -15549.371} C_VEL
LIN {X 0,Y 318.126,Z 323.042,A -85,B 0,C 180,E1 -15550.144,E2 -15550.144} C_VEL
LIN {X 0,Y 317.109,Z 334.2,A -85,B 0,C 180,E1 -15551.087,E2 -15551.087} C_VEL
LIN {X 0,Y 315.765,Z 345.833,A -85,B 0,C 180,E1 -15552.347,E2 -15552.347} C_VEL
LIN {X 0,Y 314.615,Z 356.812,A -85,B 0,C 180,E1 -15553.855,E2 -15553.855} C_VEL
LIN {X 0,Y 313.6,Z 365.826,A -85,B 0,C 180,E1 -15555.397,E2 -15555.397} C_VEL
LIN {X 0,Y 312.512,Z 374.969,A -85,B 0,C 180,E1 -15557.334,E2 -15557.334} C_VEL
LIN {X 0,Y 311.712,Z 382.319,A -85,B 0,C 180,E1 -15559.28,E2 -15559.28} C_VEL
LIN {X 0,Y 311.255,Z 387.262,A -85,B 0,C 180,E1 -15560.906,E2 -15560.906} C_VEL
LIN {X 0,Y 310.925,Z 392.044,A -85,B 0,C 180,E1 -15562.858,E2 -15562.858} C_VEL
LIN {X 0,Y 310.746,Z 395.664,A -85,B 0,C 180,E1 -15564.809,E2 -15564.809} C_VEL
LIN {X 0,Y 310.719,Z 397.496,A -85,B 0,C 180,E1 -15566.109,E2 -15566.109} C_VEL
LIN {X 0,Y 310.683,Z 398.858,A -85,B 0,C 180,E1 -15567.407,E2 -15567.407} C_VEL
LIN {X 0,Y 310.66,Z 399.81,A -85,B 0,C 180,E1 -15568.704,E2 -15568.704} C_VEL
LIN {X 0,Y 310.693,Z 400.36,A -85,B 0,C 180,E1 -15570,E2 -15570} C_VEL
LIN {X 0,Y 310.649,Z 400.461,A -85,B 0,C 180,E1 -15571.296,E2 -15571.296} C_VEL
LIN {X 0,Y 310.677,Z 400.147,A -85,B 0,C 180,E1 -15572.593,E2 -15572.593} C_VEL
LIN {X 0,Y 310.696,Z 399.439,A -85,B 0,C 180,E1 -15573.891,E2 -15573.891} C_VEL
LIN {X 0,Y 310.726,Z 397.853,A -85,B 0,C 180,E1 -15575.615,E2 -15575.615} C_VEL
LIN {X 0,Y 311.044,Z 394.778,A -85,B 0,C 180,E1 -15577.791,E2 -15577.791} C_VEL
LIN {X 0,Y 311.566,Z 390.936,A -85,B 0,C 180,E1 -15579.74,E2 -15579.74} C_VEL
LIN {X 0,Y 312.358,Z 385.967,A -85,B 0,C 180,E1 -15581.683,E2 -15581.683} C_VEL
LIN {X 0,Y 313.432,Z 379.727,A -85,B 0,C 180,E1 -15583.617,E2 -15583.617} C_VEL
LIN {X 0,Y 314.988,Z 371.988,A -85,B 0,C 180,E1 -15585.53,E2 -15585.53} C_VEL
LIN {X 0,Y 316.301,Z 363.396,A -85,B 0,C 180,E1 -15587.254,E2 -15587.254} C_VEL
LIN {X 0,Y 318.036,Z 353.481,A -85,B 0,C 180,E1 -15588.855,E2 -15588.855} C_VEL
LIN {X 0,Y 319.91,Z 342.713,A -85,B 0,C 180,E1 -15590.243,E2 -15590.243} C_VEL
LIN {X 0,Y 321.608,Z 330.588,A -85,B 0,C 180,E1 -15591.471,E2 -15591.471} C_VEL
LIN {X 0,Y 323.169,Z 317.783,A -85,B 0,C 180,E1 -15592.453,E2 -15592.453} C_VEL
LIN {X 0,Y 324.342,Z 305.667,A -85,B 0,C 180,E1 -15593.125,E2 -15593.125} C_VEL
LIN {X 0,Y 325.258,Z 292.467,A -85,B 0,C 180,E1 -15593.603,E2 -15593.603} C_VEL
LIN {X 0,Y 327.342,Z 228.637,A -85,B 0,C 180,E1 -15595.236,E2 -15595.236} C_VEL
LIN {X 0,Y 324.205,Z 208.984,A -85,B 0,C 180,E1 -15596.156,E2 -15596.156} C_VEL
LIN {X 0,Y 321.028,Z 194.66,A -85,B 0,C 180,E1 -15596.95,E2 -15596.95} C_VEL
LIN {X 0,Y 318.626,Z 189.199,A -85,B 0,C 180,E1 -15597.402,E2 -15597.402} C_VEL
LIN {X 0,Y 317.713,Z 186.817,A -85,B 0,C 180,E1 -15597.605,E2 -15597.605} C_VEL
LIN {X 0,Y 316.136,Z 178.705,A -85,B 0,C 180,E1 -15600.214,E2 -15600.214} C_VEL
LIN {X 0,Y 313.932,Z 170.045,A -85,B 0,C 180,E1 -15603.217,E2 -15603.217} C_VEL
LIN {X 0,Y 312.536,Z 164.554,A -85,B 0,C 180,E1 -15605.283,E2 -15605.283} C_VEL
LIN {X 0,Y 312.463,Z 164.567,A -85,B 0,C 180,E1 -15609.033,E2 -15609.033} C_VEL
LIN {X 0,Y 312.462,Z 164.565,A -85,B 0,C 180,E1 -15612.435,E2 -15612.435} C_VEL
LIN {X 0,Y 312.454,Z 164.566,A -85,B 0,C 180,E1 -15616.035,E2 -15616.035} C_VEL
LIN {X 0,Y 312.452,Z 164.561,A -85,B 0,C 180,E1 -15619.885,E2 -15619.885} C_VEL
LIN {X 0,Y 312.53,Z 164.549,A -85,B 0,C 180,E1 -15624.05,E2 -15624.05} C_VEL
LIN {X 0,Y 312.498,Z 164.554,A -85,B 0,C 180,E1 -15627.333,E2 -15627.333} C_VEL
LIN {X 0,Y 312.493,Z 164.558,A -85,B 0,C 180,E1 -15631.294,E2 -15631.294} C_VEL
LIN {X 0,Y 312.516,Z 164.553,A -85,B 0,C 180,E1 -15634.704,E2 -15634.704} C_VEL
LIN {X 0,Y 312.534,Z 164.544,A -85,B 0,C 180,E1 -15637.524,E2 -15637.524} C_VEL
LIN {X 0,Y 312.535,Z 164.546,A -85,B 0,C 180,E1 -15641.65,E2 -15641.65} C_VEL
LIN {X 0,Y 312.645,Z 164.535,A -85,B 0,C 180,E1 -15645.683,E2 -15645.683} C_VEL
LIN {X 0,Y 312.678,Z 164.535,A -85,B 0,C 180,E1 -15649.641,E2 -15649.641} C_VEL
LIN {X 0,Y 312.789,Z 164.517,A -85,B 0,C 180,E1 -15652.252,E2 -15652.252} C_VEL
LIN {X 0,Y 312.677,Z 164.529,A -85,B 0,C 180,E1 -15654.841,E2 -15654.841} C_VEL
LIN {X 0,Y 312.96,Z 164.5,A -85,B 0,C 180,E1 -15658.713,E2 -15658.713} C_VEL
LIN {X 0,Y 312.96,Z 164.498,A -85,B 0,C 180,E1 -15661.286,E2 -15661.286} C_VEL
LIN {X 0,Y 312.678,Z 164.536,A -85,B 0,C 180,E1 -15665.158,E2 -15665.158} C_VEL
LIN {X 0,Y 312.788,Z 164.522,A -85,B 0,C 180,E1 -15667.747,E2 -15667.747} C_VEL
LIN {X 0,Y 312.652,Z 164.546,A -85,B 0,C 180,E1 -15671.671,E2 -15671.671} C_VEL
LIN {X 0,Y 312.654,Z 164.71,A -85,B 0,C 180,E1 -15672.824,E2 -15672.824} C_VEL
LIN {X 0,Y 314.905,Z 173.595,A -85,B 0,C 180,E1 -15676.115,E2 -15676.115} C_VEL
LIN {X 0,Y 322.653,Z 189.452,A -85,B 0,C 180,E1 -15677.55,E2 -15677.55} C_VEL
LIN {X 0,Y 327.012,Z 200.083,A -85,B 0,C 180,E1 -15678.359,E2 -15678.359} C_VEL
LIN {X 0,Y 328.125,Z 206.076,A -85,B 0,C 180,E1 -15678.659,E2 -15678.659} C_VEL
LIN {X 0,Y 325.31,Z 281.693,A -85,B 0,C 180,E1 -15680.597,E2 -15680.597} C_VEL
LIN {X 0,Y 324.409,Z 295.015,A -85,B 0,C 180,E1 -15681.186,E2 -15681.186} C_VEL
LIN {X 0,Y 323.366,Z 306.719,A -85,B 0,C 180,E1 -15681.934,E2 -15681.934} C_VEL
LIN {X 0,Y 321.926,Z 318.833,A -85,B 0,C 180,E1 -15682.968,E2 -15682.968} C_VEL
LIN {X 0,Y 320.443,Z 329.359,A -85,B 0,C 180,E1 -15684.119,E2 -15684.119} C_VEL
LIN {X 0,Y 318.777,Z 339.34,A -85,B 0,C 180,E1 -15685.469,E2 -15685.469} C_VEL
LIN {X 0,Y 317.209,Z 348.544,A -85,B 0,C 180,E1 -15687.012,E2 -15687.012} C_VEL
LIN {X 0,Y 315.78,Z 356.22,A -85,B 0,C 180,E1 -15688.587,E2 -15688.587} C_VEL
LIN {X 0,Y 314.248,Z 364.11,A -85,B 0,C 180,E1 -15690.593,E2 -15690.593} C_VEL
LIN {X 0,Y 313.086,Z 370.336,A -85,B 0,C 180,E1 -15692.597,E2 -15692.597} C_VEL
LIN {X 0,Y 312.321,Z 374.387,A -85,B 0,C 180,E1 -15694.233,E2 -15694.233} C_VEL
LIN {X 0,Y 311.704,Z 377.687,A -85,B 0,C 180,E1 -15695.889,E2 -15695.889} C_VEL
LIN {X 0,Y 311.163,Z 380.49,A -85,B 0,C 180,E1 -15697.767,E2 -15697.767} C_VEL
LIN {X 0,Y 310.769,Z 382.449,A -85,B 0,C 180,E1 -15699.746,E2 -15699.746} C_VEL
LIN {X 0,Y 310.523,Z 383.43,A -85,B 0,C 180,E1 -15701.68,E2 -15701.68} C_VEL
LIN {X 0,Y 310.407,Z 383.518,A -85,B 0,C 180,E1 -15703.572,E2 -15703.572} C_VEL
LIN {X 0,Y 310.436,Z 382.769,A -85,B 0,C 180,E1 -15705.429,E2 -15705.429} C_VEL
LIN {X 0,Y 310.585,Z 381.229,A -85,B 0,C 180,E1 -15707.247,E2 -15707.247} C_VEL
LIN {X 0,Y 310.881,Z 377.857,A -85,B 0,C 180,E1 -15709.656,E2 -15709.656} C_VEL
LIN {X 0,Y 311.289,Z 374.163,A -85,B 0,C 180,E1 -15711.515,E2 -15711.515} C_VEL
LIN {X 0,Y 311.899,Z 368.37,A -85,B 0,C 180,E1 -15713.738,E2 -15713.738} C_VEL
LIN {X 0,Y 312.674,Z 361.333,A -85,B 0,C 180,E1 -15715.812,E2 -15715.812} C_VEL
LIN {X 0,Y 313.615,Z 353.384,A -85,B 0,C 180,E1 -15717.678,E2 -15717.678} C_VEL
LIN {X 0,Y 314.717,Z 344.244,A -85,B 0,C 180,E1 -15719.414,E2 -15719.414} C_VEL
LIN {X 0,Y 315.761,Z 334.817,A -85,B 0,C 180,E1 -15720.865,E2 -15720.865} C_VEL
LIN {X 0,Y 317.003,Z 323.544,A -85,B 0,C 180,E1 -15722.253,E2 -15722.253} C_VEL
LIN {X 0,Y 318.071,Z 311.554,A -85,B 0,C 180,E1 -15723.421,E2 -15723.421} C_VEL
LIN {X 0,Y 319.054,Z 299.242,A -85,B 0,C 180,E1 -15724.319,E2 -15724.319} C_VEL
LIN {X 0,Y 319.755,Z 285.542,A -85,B 0,C 180,E1 -15725.036,E2 -15725.036} C_VEL
LIN {X 0,Y 320.282,Z 272.683,A -85,B 0,C 180,E1 -15725.447,E2 -15725.447} C_VEL
LIN {X 0,Y 322.05,Z 202.728,A -85,B 0,C 180,E1 -15727.169,E2 -15727.169} C_VEL
LIN {X 0,Y 319.2,Z 187.408,A -85,B 0,C 180,E1 -15727.756,E2 -15727.756} C_VEL
LIN {X 0,Y 314.107,Z 172.354,A -85,B 0,C 180,E1 -15728.508,E2 -15728.508} C_VEL
LIN {X 0,Y 312.583,Z 164.55,A -85,B 0,C 180,E1 -15731.05,E2 -15731.05} C_VEL
LIN {X 0,Y 312.647,Z 164.539,A -85,B 0,C 180,E1 -15735.684,E2 -15735.684} C_VEL
LIN {X 0,Y 312.68,Z 164.534,A -85,B 0,C 180,E1 -15739.641,E2 -15739.641} C_VEL
LIN {X 0,Y 312.793,Z 164.524,A -85,B 0,C 180,E1 -15742.253,E2 -15742.253} C_VEL
LIN {X 0,Y 312.683,Z 164.534,A -85,B 0,C 180,E1 -15744.842,E2 -15744.842} C_VEL
LIN {X 0,Y 312.963,Z 164.499,A -85,B 0,C 180,E1 -15748.713,E2 -15748.713} C_VEL
LIN {X 0,Y 312.962,Z 164.499,A -85,B 0,C 180,E1 -15751.287,E2 -15751.287} C_VEL
LIN {X 0,Y 312.681,Z 164.534,A -85,B 0,C 180,E1 -15755.158,E2 -15755.158} C_VEL
LIN {X 0,Y 312.792,Z 164.523,A -85,B 0,C 180,E1 -15757.748,E2 -15757.748} C_VEL
LIN {X 0,Y 312.656,Z 164.541,A -85,B 0,C 180,E1 -15761.672,E2 -15761.672} C_VEL
LIN {X 0,Y 312.61,Z 164.542,A -85,B 0,C 180,E1 -15764.828,E2 -15764.828} C_VEL
LIN {X 0,Y 312.531,Z 164.553,A -85,B 0,C 180,E1 -15769.186,E2 -15769.186} C_VEL
LIN {X 0,Y 312.51,Z 164.555,A -85,B 0,C 180,E1 -15772.775,E2 -15772.775} C_VEL
LIN {X 0,Y 312.478,Z 164.559,A -85,B 0,C 180,E1 -15776.732,E2 -15776.732} C_VEL
LIN {X 0,Y 312.464,Z 164.563,A -85,B 0,C 180,E1 -15779.658,E2 -15779.658} C_VEL
LIN {X 0,Y 312.516,Z 164.556,A -85,B 0,C 180,E1 -15783.689,E2 -15783.689} C_VEL
LIN {X 0,Y 312.509,Z 164.559,A -85,B 0,C 180,E1 -15787.387,E2 -15787.387} C_VEL
LIN {X 0,Y 312.436,Z 164.565,A -85,B 0,C 180,E1 -15790.717,E2 -15790.717} C_VEL
LIN {X 0,Y 312.445,Z 164.561,A -85,B 0,C 180,E1 -15794.21,E2 -15794.21} C_VEL
LIN {X 0,Y 312.449,Z 164.562,A -85,B 0,C 180,E1 -15797.412,E2 -15797.412} C_VEL
LIN {X 0,Y 311.825,Z 164.644,A -85,B 0,C 180,E1 -15798.488,E2 -15798.488} C_VEL
LIN {X 0,Y 308.955,Z 164.998,A -85,B 0,C 180,E1 -15800.237,E2 -15800.237} C_VEL
LIN {X 0,Y 306.515,Z 165.301,A -85,B 0,C 180,E1 -15801.656,E2 -15801.656} C_VEL
LIN {X 0,Y 305.502,Z 165.431,A -85,B 0,C 180,E1 -15802.756,E2 -15802.756} C_VEL
LIN {X 0,Y 305.439,Z 165.435,A -85,B 0,C 180,E1 -15803.128,E2 -15803.128} C_VEL
LIN {X 0,Y 305.46,Z 165.432,A -85,B 0,C 180,E1 -15806.483,E2 -15806.483} C_VEL
LIN {X 0,Y 305.425,Z 165.436,A -85,B 0,C 180,E1 -15809.587,E2 -15809.587} C_VEL
LIN {X 0,Y 305.444,Z 165.439,A -85,B 0,C 180,E1 -15812.602,E2 -15812.602} C_VEL
LIN {X 0,Y 305.435,Z 165.436,A -85,B 0,C 180,E1 -15815.533,E2 -15815.533} C_VEL
LIN {X 0,Y 305.472,Z 165.43,A -85,B 0,C 180,E1 -15819.812,E2 -15819.812} C_VEL
LIN {X 0,Y 305.509,Z 165.426,A -85,B 0,C 180,E1 -15823.976,E2 -15823.976} C_VEL
LIN {X 0,Y 305.565,Z 165.422,A -85,B 0,C 180,E1 -15826.704,E2 -15826.704} C_VEL
LIN {X 0,Y 305.68,Z 165.406,A -85,B 0,C 180,E1 -15830.739,E2 -15830.739} C_VEL
LIN {X 0,Y 305.779,Z 165.391,A -85,B 0,C 180,E1 -15833.402,E2 -15833.402} C_VEL
LIN {X 0,Y 305.929,Z 165.375,A -85,B 0,C 180,E1 -15838.684,E2 -15838.684} C_VEL
LIN {X 0,Y 305.929,Z 165.374,A -85,B 0,C 180,E1 -15841.317,E2 -15841.317} C_VEL
LIN {X 0,Y 305.78,Z 165.391,A -85,B 0,C 180,E1 -15846.6,E2 -15846.6} C_VEL
LIN {X 0,Y 305.681,Z 165.405,A -85,B 0,C 180,E1 -15849.262,E2 -15849.262} C_VEL
LIN {X 0,Y 305.566,Z 165.421,A -85,B 0,C 180,E1 -15853.298,E2 -15853.298} C_VEL
LIN {X 0,Y 305.502,Z 165.428,A -85,B 0,C 180,E1 -15856.026,E2 -15856.026} C_VEL
LIN {X 0,Y 305.47,Z 165.433,A -85,B 0,C 180,E1 -15860.189,E2 -15860.189} C_VEL
LIN {X 0,Y 305.436,Z 165.435,A -85,B 0,C 180,E1 -15864.468,E2 -15864.468} C_VEL
LIN {X 0,Y 305.438,Z 165.441,A -85,B 0,C 180,E1 -15867.4,E2 -15867.4} C_VEL
LIN {X 0,Y 305.415,Z 165.438,A -85,B 0,C 180,E1 -15870.415,E2 -15870.415} C_VEL
LIN {X 0,Y 305.463,Z 165.431,A -85,B 0,C 180,E1 -15874.079,E2 -15874.079} C_VEL
LIN {X 0,Y 305.452,Z 165.435,A -85,B 0,C 180,E1 -15876.743,E2 -15876.743} C_VEL
